LIN {X 0,Y 263.133,Z 902.515,A -85,B 0,C 180,E1 -18302.289,E2 -18302.289} C_VEL
LIN {X 0,Y 263.178,Z 902.512,A -85,B 0,C 180,E1 -18306.76,E2 -18306.76} C_VEL
LIN {X 0,Y 263.095,Z 902.525,A -85,B 0,C 180,E1 -18309.875,E2 -18309.875} C_VEL
LIN {X 0,Y 263.08,Z 902.529,A -85,B 0,C 180,E1 -18313.994,E2 -18313.994} C_VEL
LIN {X 0,Y 263.112,Z 902.522,A -85,B 0,C 180,E1 -18318.41,E2 -18318.41} C_VEL
LIN {X 0,Y 263.133,Z 902.519,A -85,B 0,C 180,E1 -18322.098,E2 -18322.098} C_VEL
LIN {X 0,Y 263.155,Z 902.516,A -85,B 0,C 180,E1 -18325.885,E2 -18325.885} C_VEL
LIN {X 0,Y 263.129,Z 902.516,A -85,B 0,C 180,E1 -18329.503,E2 -18329.503} C_VEL
LIN {X 0,Y 263.13,Z 902.521,A -85,B 0,C 180,E1 -18332.995,E2 -18332.995} C_VEL
LIN {X 0,Y 263.118,Z 902.52,A -85,B 0,C 180,E1 -18336.38,E2 -18336.38} C_VEL
LIN {X 0,Y 263.21,Z 902.507,A -85,B 0,C 180,E1 -18339.688,E2 -18339.688} C_VEL
LIN {X 0,Y 263.292,Z 902.498,A -85,B 0,C 180,E1 -18344.518,E2 -18344.518} C_VEL
LIN {X 0,Y 263.334,Z 902.493,A -85,B 0,C 180,E1 -18349.232,E2 -18349.232} C_VEL
LIN {X 0,Y 263.529,Z 902.469,A -85,B 0,C 180,E1 -18352.336,E2 -18352.336} C_VEL
LIN {X 0,Y 263.726,Z 902.443,A -85,B 0,C 180,E1 -18358.472,E2 -18358.472} C_VEL
LIN {X 0,Y 263.726,Z 902.445,A -85,B 0,C 180,E1 -18361.526,E2 -18361.526} C_VEL
LIN {X 0,Y 263.528,Z 902.467,A -85,B 0,C 180,E1 -18367.662,E2 -18367.662} C_VEL
LIN {X 0,Y 263.345,Z 902.494,A -85,B 0,C 180,E1 -18370.766,E2 -18370.766} C_VEL
LIN {X 0,Y 263.29,Z 902.496,A -85,B 0,C 180,E1 -18375.481,E2 -18375.481} C_VEL
LIN {X 0,Y 263.208,Z 902.509,A -85,B 0,C 180,E1 -18380.31,E2 -18380.31} C_VEL
LIN {X 0,Y 263.126,Z 902.52,A -85,B 0,C 180,E1 -18385.299,E2 -18385.299} C_VEL
LIN {X 0,Y 263.132,Z 902.518,A -85,B 0,C 180,E1 -18388.738,E2 -18388.738} C_VEL
LIN {X 0,Y 262.413,Z 902.609,A -85,B 0,C 180,E1 -18390.015,E2 -18390.015} C_VEL
LIN {X 0,Y 259.57,Z 902.961,A -85,B 0,C 180,E1 -18392.099,E2 -18392.099} C_VEL
LIN {X 0,Y 257.184,Z 903.26,A -85,B 0,C 180,E1 -18393.793,E2 -18393.793} C_VEL
LIN {X 0,Y 256.155,Z 903.386,A -85,B 0,C 180,E1 -18395.105,E2 -18395.105} C_VEL
LIN {X 0,Y 256.065,Z 903.395,A -85,B 0,C 180,E1 -18395.55,E2 -18395.55} C_VEL
LIN {X 0,Y 256.066,Z 903.399,A -85,B 0,C 180,E1 -18399.142,E2 -18399.142} C_VEL
LIN {X 0,Y 256.028,Z 903.402,A -85,B 0,C 180,E1 -18403.334,E2 -18403.334} C_VEL
LIN {X 0,Y 256.055,Z 903.402,A -85,B 0,C 180,E1 -18407.822,E2 -18407.822} C_VEL
LIN {X 0,Y 256.065,Z 903.398,A -85,B 0,C 180,E1 -18410.856,E2 -18410.856} C_VEL
LIN {X 0,Y 256.12,Z 903.39,A -85,B 0,C 180,E1 -18412.865,E2 -18412.865} C_VEL
LIN {X 0,Y 256.065,Z 903.401,A -85,B 0,C 180,E1 -18416.706,E2 -18416.706} C_VEL
LIN {X 0,Y 256.251,Z 903.416,A -85,B 0,C 180,E1 -18421.718,E2 -18421.718} C_VEL
LIN {X 0,Y 258.143,Z 913.925,A -85,B 0,C 180,E1 -18425.897,E2 -18425.897} C_VEL
LIN {X 0,Y 257.046,Z 922.563,A -85,B 0,C 180,E1 -18429.179,E2 -18429.179} C_VEL
LIN {X 0,Y 256.802,Z 924.586,A -85,B 0,C 180,E1 -18429.943,E2 -18429.943} C_VEL
LIN {X 0,Y 257.654,Z 940.89,A -85,B 0,C 180,E1 -18430.712,E2 -18430.712} C_VEL
LIN {X 0,Y 259.789,Z 963.766,A -85,B 0,C 180,E1 -18431.766,E2 -18431.766} C_VEL
LIN {X 0,Y 258.613,Z 1004.147,A -85,B 0,C 180,E1 -18433.572,E2 -18433.572} C_VEL
LIN {X 0,Y 257.814,Z 1016.929,A -85,B 0,C 180,E1 -18434.485,E2 -18434.485} C_VEL
LIN {X 0,Y 257.36,Z 1025.939,A -85,B 0,C 180,E1 -18435.368,E2 -18435.368} C_VEL
LIN {X 0,Y 256.718,Z 1035.432,A -85,B 0,C 180,E1 -18436.544,E2 -18436.544} C_VEL
LIN {X 0,Y 255.948,Z 1045.484,A -85,B 0,C 180,E1 -18438.115,E2 -18438.115} C_VEL
LIN {X 0,Y 255.437,Z 1053.431,A -85,B 0,C 180,E1 -18439.698,E2 -18439.698} C_VEL
LIN {X 0,Y 255.026,Z 1059.956,A -85,B 0,C 180,E1 -18441.282,E2 -18441.282} C_VEL
LIN {X 0,Y 254.757,Z 1065.381,A -85,B 0,C 180,E1 -18442.869,E2 -18442.869} C_VEL
LIN {X 0,Y 254.53,Z 1070.615,A -85,B 0,C 180,E1 -18444.755,E2 -18444.755} C_VEL
LIN {X 0,Y 254.336,Z 1075.116,A -85,B 0,C 180,E1 -18446.832,E2 -18446.832} C_VEL
LIN {X 0,Y 254.233,Z 1078.877,A -85,B 0,C 180,E1 -18449.208,E2 -18449.208} C_VEL
LIN {X 0,Y 254.094,Z 1081.168,A -85,B 0,C 180,E1 -18451.585,E2 -18451.585} C_VEL
LIN {X 0,Y 254.152,Z 1082.036,A -85,B 0,C 180,E1 -18453.17,E2 -18453.17} C_VEL
LIN {X 0,Y 254.131,Z 1082.299,A -85,B 0,C 180,E1 -18455.394,E2 -18455.394} C_VEL
LIN {X 0,Y 254.574,Z 1081.302,A -85,B 0,C 180,E1 -18457.934,E2 -18457.934} C_VEL
LIN {X 0,Y 255.122,Z 1080.076,A -85,B 0,C 180,E1 -18459.514,E2 -18459.514} C_VEL
LIN {X 0,Y 256.305,Z 1077.127,A -85,B 0,C 180,E1 -18461.867,E2 -18461.867} C_VEL
LIN {X 0,Y 257.32,Z 1074.54,A -85,B 0,C 180,E1 -18463.424,E2 -18463.424} C_VEL
LIN {X 0,Y 259.264,Z 1069.361,A -85,B 0,C 180,E1 -18465.728,E2 -18465.728} C_VEL
LIN {X 0,Y 261.247,Z 1063.88,A -85,B 0,C 180,E1 -18467.616,E2 -18467.616} C_VEL
LIN {X 0,Y 263.629,Z 1057.201,A -85,B 0,C 180,E1 -18469.465,E2 -18469.465} C_VEL
LIN {X 0,Y 266.42,Z 1048.971,A -85,B 0,C 180,E1 -18471.267,E2 -18471.267} C_VEL
LIN {X 0,Y 269.478,Z 1038.482,A -85,B 0,C 180,E1 -18473.029,E2 -18473.029} C_VEL
LIN {X 0,Y 272.034,Z 1029.452,A -85,B 0,C 180,E1 -18474.213,E2 -18474.213} C_VEL
LIN {X 0,Y 274.778,Z 1018.129,A -85,B 0,C 180,E1 -18475.367,E2 -18475.367} C_VEL
LIN {X 0,Y 276.831,Z 1007.471,A -85,B 0,C 180,E1 -18476.174,E2 -18476.174} C_VEL
LIN {X 0,Y 278.749,Z 994.655,A -85,B 0,C 180,E1 -18476.888,E2 -18476.888} C_VEL
LIN {X 0,Y 281.525,Z 969.653,A -85,B 0,C 180,E1 -18478.087,E2 -18478.087} C_VEL
LIN {X 0,Y 280.837,Z 960.401,A -85,B 0,C 180,E1 -18478.98,E2 -18478.98} C_VEL
LIN {X 0,Y 279.732,Z 952.159,A -85,B 0,C 180,E1 -18479.995,E2 -18479.995} C_VEL
LIN {X 0,Y 277.278,Z 946.159,A -85,B 0,C 180,E1 -18481.289,E2 -18481.289} C_VEL
LIN {X 0,Y 275.212,Z 941.618,A -85,B 0,C 180,E1 -18482.475,E2 -18482.475} C_VEL
LIN {X 0,Y 272.839,Z 936.693,A -85,B 0,C 180,E1 -18483.982,E2 -18483.982} C_VEL
LIN {X 0,Y 270.146,Z 931.863,A -85,B 0,C 180,E1 -18485.901,E2 -18485.901} C_VEL
LIN {X 0,Y 269.36,Z 930.385,A -85,B 0,C 180,E1 -18486.552,E2 -18486.552} C_VEL
LIN {X 0,Y 265.947,Z 924.786,A -85,B 0,C 180,E1 -18490.207,E2 -18490.207} C_VEL
LIN {X 0,Y 265.122,Z 922.952,A -85,B 0,C 180,E1 -18491.764,E2 -18491.764} C_VEL
LIN {X 0,Y 264.299,Z 921.573,A -85,B 0,C 180,E1 -18494.549,E2 -18494.549} C_VEL
LIN {X 0,Y 264.876,Z 921.163,A -85,B 0,C 180,E1 -18497.981,E2 -18497.981} C_VEL
LIN {X 0,Y 267.039,Z 924.13,A -85,B 0,C 180,E1 -18501.686,E2 -18501.686} C_VEL
LIN {X 0,Y 268.847,Z 925.751,A -85,B 0,C 180,E1 -18503.356,E2 -18503.356} C_VEL
LIN {X 0,Y 271.774,Z 929.696,A -85,B 0,C 180,E1 -18505.647,E2 -18505.647} C_VEL
LIN {X 0,Y 275.456,Z 935.246,A -85,B 0,C 180,E1 -18507.921,E2 -18507.921} C_VEL
LIN {X 0,Y 278.032,Z 939.659,A -85,B 0,C 180,E1 -18509.312,E2 -18509.312} C_VEL
LIN {X 0,Y 281.299,Z 945.577,A -85,B 0,C 180,E1 -18510.871,E2 -18510.871} C_VEL
LIN {X 0,Y 283.341,Z 950.251,A -85,B 0,C 180,E1 -18511.833,E2 -18511.833} C_VEL
LIN {X 0,Y 278.626,Z 988.353,A -85,B 0,C 180,E1 -18513.655,E2 -18513.655} C_VEL
LIN {X 0,Y 276.931,Z 999.245,A -85,B 0,C 180,E1 -18514.442,E2 -18514.442} C_VEL
LIN {X 0,Y 274.839,Z 1009.763,A -85,B 0,C 180,E1 -18515.448,E2 -18515.448} C_VEL
LIN {X 0,Y 272.517,Z 1019.531,A -85,B 0,C 180,E1 -18516.641,E2 -18516.641} C_VEL
LIN {X 0,Y 269.795,Z 1029.32,A -85,B 0,C 180,E1 -18518.211,E2 -18518.211} C_VEL
LIN {X 0,Y 267.014,Z 1038.1,A -85,B 0,C 180,E1 -18519.992,E2 -18519.992} C_VEL
LIN {X 0,Y 264.523,Z 1045.179,A -85,B 0,C 180,E1 -18521.81,E2 -18521.81} C_VEL
LIN {X 0,Y 262.291,Z 1050.771,A -85,B 0,C 180,E1 -18523.66,E2 -18523.66} C_VEL
LIN {X 0,Y 260.607,Z 1054.482,A -85,B 0,C 180,E1 -18525.156,E2 -18525.156} C_VEL
LIN {X 0,Y 258.571,Z 1058.706,A -85,B 0,C 180,E1 -18527.442,E2 -18527.442} C_VEL
LIN {X 0,Y 257.501,Z 1060.839,A -85,B 0,C 180,E1 -18528.987,E2 -18528.987} C_VEL
LIN {X 0,Y 256.624,Z 1062.359,A -85,B 0,C 180,E1 -18530.543,E2 -18530.543} C_VEL
LIN {X 0,Y 255.786,Z 1063.32,A -85,B 0,C 180,E1 -18532.104,E2 -18532.104} C_VEL
LIN {X 0,Y 255.092,Z 1063.796,A -85,B 0,C 180,E1 -18533.674,E2 -18533.674} C_VEL
LIN {X 0,Y 254.684,Z 1063.773,A -85,B 0,C 180,E1 -18535.252,E2 -18535.252} C_VEL
LIN {X 0,Y 254.42,Z 1063.24,A -85,B 0,C 180,E1 -18536.834,E2 -18536.834} C_VEL
LIN {X 0,Y 254.211,Z 1062.102,A -85,B 0,C 180,E1 -18538.417,E2 -18538.417} C_VEL
LIN {X 0,Y 254.09,Z 1059.449,A -85,B 0,C 180,E1 -18540.793,E2 -18540.793} C_VEL
LIN {X 0,Y 254.195,Z 1055.35,A -85,B 0,C 180,E1 -18543.171,E2 -18543.171} C_VEL
LIN {X 0,Y 254.272,Z 1050.813,A -85,B 0,C 180,E1 -18545.152,E2 -18545.152} C_VEL
LIN {X 0,Y 254.649,Z 1045.089,A -85,B 0,C 180,E1 -18547.135,E2 -18547.135} C_VEL
LIN {X 0,Y 255.093,Z 1037.972,A -85,B 0,C 180,E1 -18549.116,E2 -18549.116} C_VEL
LIN {X 0,Y 255.772,Z 1028.878,A -85,B 0,C 180,E1 -18551.09,E2 -18551.09} C_VEL
LIN {X 0,Y 256.352,Z 1021.061,A -85,B 0,C 180,E1 -18552.469,E2 -18552.469} C_VEL
LIN {X 0,Y 256.929,Z 1012.996,A -85,B 0,C 180,E1 -18553.647,E2 -18553.647} C_VEL
LIN {X 0,Y 257.62,Z 1003.027,A -85,B 0,C 180,E1 -18554.819,E2 -18554.819} C_VEL
LIN {X 0,Y 258.247,Z 990.644,A -85,B 0,C 180,E1 -18555.894,E2 -18555.894} C_VEL
LIN {X 0,Y 258.556,Z 981.199,A -85,B 0,C 180,E1 -18556.483,E2 -18556.483} C_VEL
LIN {X 0,Y 260.259,Z 930.177,A -85,B 0,C 180,E1 -18558.702,E2 -18558.702} C_VEL
LIN {X 0,Y 256.449,Z 904,A -85,B 0,C 180,E1 -18559.967,E2 -18559.967} C_VEL
LIN {X 0,Y 256.371,Z 903.35,A -85,B 0,C 180,E1 -18560.354,E2 -18560.354} C_VEL
LIN {X 0,Y 256.075,Z 903.397,A -85,B 0,C 180,E1 -18566.049,E2 -18566.049} C_VEL
LIN {X 0,Y 256.056,Z 903.399,A -85,B 0,C 180,E1 -18569.608,E2 -18569.608} C_VEL
LIN {X 0,Y 256.068,Z 903.401,A -85,B 0,C 180,E1 -18573.294,E2 -18573.294} C_VEL
LIN {X 0,Y 256.088,Z 903.397,A -85,B 0,C 180,E1 -18577.263,E2 -18577.263} C_VEL
LIN {X 0,Y 256.011,Z 903.404,A -85,B 0,C 180,E1 -18581.213,E2 -18581.213} C_VEL
LIN {X 0,Y 256.02,Z 903.405,A -85,B 0,C 180,E1 -18585.54,E2 -18585.54} C_VEL
LIN {X 0,Y 256.041,Z 903.4,A -85,B 0,C 180,E1 -18588.794,E2 -18588.794} C_VEL
LIN {X 0,Y 256.124,Z 903.392,A -85,B 0,C 180,E1 -18592.867,E2 -18592.867} C_VEL
LIN {X 0,Y 256.069,Z 903.398,A -85,B 0,C 180,E1 -18596.708,E2 -18596.708} C_VEL
LIN {X 0,Y 256.058,Z 903.401,A -85,B 0,C 180,E1 -18600.393,E2 -18600.393} C_VEL
LIN {X 0,Y 256.136,Z 903.393,A -85,B 0,C 180,E1 -18604.889,E2 -18604.889} C_VEL
LIN {X 0,Y 256.128,Z 903.394,A -85,B 0,C 180,E1 -18609.102,E2 -18609.102} C_VEL
LIN {X 0,Y 256.233,Z 903.376,A -85,B 0,C 180,E1 -18614.081,E2 -18614.081} C_VEL
LIN {X 0,Y 256.291,Z 903.37,A -85,B 0,C 180,E1 -18618.933,E2 -18618.933} C_VEL
LIN {X 0,Y 256.494,Z 903.346,A -85,B 0,C 180,E1 -18622.126,E2 -18622.126} C_VEL
LIN {X 0,Y 256.422,Z 903.352,A -85,B 0,C 180,E1 -18626.858,E2 -18626.858} C_VEL
LIN {X 0,Y 256.69,Z 903.321,A -85,B 0,C 180,E1 -18628.431,E2 -18628.431} C_VEL
LIN {X 0,Y 256.689,Z 903.321,A -85,B 0,C 180,E1 -18631.569,E2 -18631.569} C_VEL
LIN {X 0,Y 256.457,Z 903.352,A -85,B 0,C 180,E1 -18636.294,E2 -18636.294} C_VEL
LIN {X 0,Y 256.407,Z 903.355,A -85,B 0,C 180,E1 -18639.466,E2 -18639.466} C_VEL
LIN {X 0,Y 256.208,Z 903.38,A -85,B 0,C 180,E1 -18644.293,E2 -18644.293} C_VEL
LIN {X 0,Y 256.15,Z 903.388,A -85,B 0,C 180,E1 -18647.567,E2 -18647.567} C_VEL
LIN {X 0,Y 256.124,Z 903.393,A -85,B 0,C 180,E1 -18651.097,E2 -18651.097} C_VEL
LIN {X 0,Y 256.089,Z 903.398,A -85,B 0,C 180,E1 -18655.089,E2 -18655.089} C_VEL
LIN {X 0,Y 256.094,Z 903.395,A -85,B 0,C 180,E1 -18658.575,E2 -18658.575} C_VEL
LIN {X 0,Y 256.078,Z 903.396,A -85,B 0,C 180,E1 -18661.701,E2 -18661.701} C_VEL
LIN {X 0,Y 256.083,Z 903.397,A -85,B 0,C 180,E1 -18665.193,E2 -18665.193} C_VEL
LIN {X 0,Y 256.109,Z 903.395,A -85,B 0,C 180,E1 -18667.267,E2 -18667.267} C_VEL
LIN {X 0,Y 256.043,Z 903.399,A -85,B 0,C 180,E1 -18671.206,E2 -18671.206} C_VEL
LIN {X 0,Y 256.022,Z 903.405,A -85,B 0,C 180,E1 -18675.539,E2 -18675.539} C_VEL
LIN {X 0,Y 256.043,Z 903.4,A -85,B 0,C 180,E1 -18678.793,E2 -18678.793} C_VEL
LIN {X 0,Y 256.107,Z 903.393,A -85,B 0,C 180,E1 -18682.862,E2 -18682.862} C_VEL
LIN {X 0,Y 256.07,Z 903.4,A -85,B 0,C 180,E1 -18686.707,E2 -18686.707} C_VEL
LIN {X 0,Y 256.058,Z 903.399,A -85,B 0,C 180,E1 -18690.392,E2 -18690.392} C_VEL
LIN {X 0,Y 256.077,Z 903.396,A -85,B 0,C 180,E1 -18693.951,E2 -18693.951} C_VEL
LIN {X 0,Y 256.06,Z 903.399,A -85,B 0,C 180,E1 -18697.402,E2 -18697.402} C_VEL
LIN {X 0,Y 256.107,Z 903.393,A -85,B 0,C 180,E1 -18700.773,E2 -18700.773} C_VEL
LIN {X 0,Y 256.217,Z 903.379,A -85,B 0,C 180,E1 -18704.079,E2 -18704.079} C_VEL
LIN {X 0,Y 256.278,Z 903.37,A -85,B 0,C 180,E1 -18708.932,E2 -18708.932} C_VEL
LIN {X 0,Y 256.493,Z 903.346,A -85,B 0,C 180,E1 -18712.125,E2 -18712.125} C_VEL
LIN {X 0,Y 256.419,Z 903.352,A -85,B 0,C 180,E1 -18716.857,E2 -18716.857} C_VEL
LIN {X 0,Y 256.688,Z 903.32,A -85,B 0,C 180,E1 -18718.43,E2 -18718.43} C_VEL
LIN {X 0,Y 256.687,Z 903.322,A -85,B 0,C 180,E1 -18721.568,E2 -18721.568} C_VEL
LIN {X 0,Y 256.454,Z 903.352,A -85,B 0,C 180,E1 -18726.293,E2 -18726.293} C_VEL
LIN {X 0,Y 256.404,Z 903.355,A -85,B 0,C 180,E1 -18729.465,E2 -18729.465} C_VEL
LIN {X 0,Y 256.205,Z 903.382,A -85,B 0,C 180,E1 -18734.292,E2 -18734.292} C_VEL
LIN {X 0,Y 256.146,Z 903.387,A -85,B 0,C 180,E1 -18737.566,E2 -18737.566} C_VEL
LIN {X 0,Y 256.12,Z 903.395,A -85,B 0,C 180,E1 -18741.096,E2 -18741.096} C_VEL
LIN {X 0,Y 256.085,Z 903.398,A -85,B 0,C 180,E1 -18745.088,E2 -18745.088} C_VEL
LIN {X 0,Y 256.08,Z 903.396,A -85,B 0,C 180,E1 -18748.716,E2 -18748.716} C_VEL
LIN {X 0,Y 256.074,Z 903.399,A -85,B 0,C 180,E1 -18751.7,E2 -18751.7} C_VEL
LIN {X 0,Y 256.065,Z 903.395,A -85,B 0,C 180,E1 -18755.55,E2 -18755.55} C_VEL
LIN {X 0,Y 255.361,Z 903.486,A -85,B 0,C 180,E1 -18756.862,E2 -18756.862} C_VEL
LIN {X 0,Y 252.442,Z 903.85,A -85,B 0,C 180,E1 -18759,E2 -18759} C_VEL
LIN {X 0,Y 250.017,Z 904.151,A -85,B 0,C 180,E1 -18760.74,E2 -18760.74} C_VEL
LIN {X 0,Y 249.034,Z 904.275,A -85,B 0,C 180,E1 -18762.092,E2 -18762.092} C_VEL
LIN {X 0,Y 248.985,Z 904.278,A -85,B 0,C 180,E1 -18762.549,E2 -18762.549} C_VEL
LIN {X 0,Y 248.992,Z 904.279,A -85,B 0,C 180,E1 -18767.357,E2 -18767.357} C_VEL
LIN {X 0,Y 249.036,Z 904.276,A -85,B 0,C 180,E1 -18772.202,E2 -18772.202} C_VEL
LIN {X 0,Y 249.042,Z 904.272,A -85,B 0,C 180,E1 -18775.639,E2 -18775.639} C_VEL
LIN {X 0,Y 249.063,Z 904.27,A -85,B 0,C 180,E1 -18779.474,E2 -18779.474} C_VEL
LIN {X 0,Y 249.221,Z 904.386,A -85,B 0,C 180,E1 -18781.755,E2 -18781.755} C_VEL
LIN {X 0,Y 251.008,Z 913.787,A -85,B 0,C 180,E1 -18785.607,E2 -18785.607} C_VEL
LIN {X 0,Y 250.576,Z 918.515,A -85,B 0,C 180,E1 -18787.467,E2 -18787.467} C_VEL
LIN {X 0,Y 249.741,Z 924.538,A -85,B 0,C 180,E1 -18789.781,E2 -18789.781} C_VEL
LIN {X 0,Y 250.582,Z 941.022,A -85,B 0,C 180,E1 -18790.561,E2 -18790.561} C_VEL
LIN {X 0,Y 252.716,Z 964.072,A -85,B 0,C 180,E1 -18791.658,E2 -18791.658} C_VEL
LIN {X 0,Y 251.522,Z 1004.006,A -85,B 0,C 180,E1 -18793.513,E2 -18793.513} C_VEL
LIN {X 0,Y 250.741,Z 1016.613,A -85,B 0,C 180,E1 -18794.453,E2 -18794.453} C_VEL
LIN {X 0,Y 250.286,Z 1025.554,A -85,B 0,C 180,E1 -18795.361,E2 -18795.361} C_VEL
LIN {X 0,Y 249.63,Z 1034.982,A -85,B 0,C 180,E1 -18796.569,E2 -18796.569} C_VEL
LIN {X 0,Y 248.895,Z 1045.021,A -85,B 0,C 180,E1 -18798.187,E2 -18798.187} C_VEL
LIN {X 0,Y 248.369,Z 1052.947,A -85,B 0,C 180,E1 -18799.813,E2 -18799.813} C_VEL
LIN {X 0,Y 247.955,Z 1059.493,A -85,B 0,C 180,E1 -18801.442,E2 -18801.442} C_VEL
LIN {X 0,Y 247.675,Z 1065.579,A -85,B 0,C 180,E1 -18803.288,E2 -18803.288} C_VEL
LIN {X 0,Y 247.481,Z 1070.445,A -85,B 0,C 180,E1 -18805.112,E2 -18805.112} C_VEL
LIN {X 0,Y 247.336,Z 1073.949,A -85,B 0,C 180,E1 -18806.742,E2 -18806.742} C_VEL
LIN {X 0,Y 247.221,Z 1076.763,A -85,B 0,C 180,E1 -18808.371,E2 -18808.371} C_VEL
LIN {X 0,Y 247.214,Z 1078.945,A -85,B 0,C 180,E1 -18810,E2 -18810} C_VEL
LIN {X 0,Y 247.029,Z 1080.482,A -85,B 0,C 180,E1 -18811.63,E2 -18811.63} C_VEL
LIN {X 0,Y 247.084,Z 1081.422,A -85,B 0,C 180,E1 -18813.261,E2 -18813.261} C_VEL
LIN {X 0,Y 247.034,Z 1081.887,A -85,B 0,C 180,E1 -18815.302,E2 -18815.302} C_VEL
LIN {X 0,Y 247.526,Z 1081.253,A -85,B 0,C 180,E1 -18818.161,E2 -18818.161} C_VEL
LIN {X 0,Y 248.109,Z 1080.109,A -85,B 0,C 180,E1 -18819.785,E2 -18819.785} C_VEL
LIN {X 0,Y 249.372,Z 1077.508,A -85,B 0,C 180,E1 -18822.202,E2 -18822.202} C_VEL
LIN {X 0,Y 251.129,Z 1073.57,A -85,B 0,C 180,E1 -18824.588,E2 -18824.588} C_VEL
LIN {X 0,Y 252.5,Z 1070.287,A -85,B 0,C 180,E1 -18826.161,E2 -18826.161} C_VEL
LIN {X 0,Y 255.068,Z 1063.948,A -85,B 0,C 180,E1 -18828.473,E2 -18828.473} C_VEL
LIN {X 0,Y 257.629,Z 1057.311,A -85,B 0,C 180,E1 -18830.353,E2 -18830.353} C_VEL
LIN {X 0,Y 260.593,Z 1049.298,A -85,B 0,C 180,E1 -18832.183,E2 -18832.183} C_VEL
LIN {X 0,Y 263.889,Z 1039.169,A -85,B 0,C 180,E1 -18833.963,E2 -18833.963} C_VEL
LIN {X 0,Y 266.569,Z 1030.293,A -85,B 0,C 180,E1 -18835.159,E2 -18835.159} C_VEL
LIN {X 0,Y 269.459,Z 1019.526,A -85,B 0,C 180,E1 -18836.32,E2 -18836.32} C_VEL
LIN {X 0,Y 272.093,Z 1007.264,A -85,B 0,C 180,E1 -18837.288,E2 -18837.288} C_VEL
LIN {X 0,Y 274.032,Z 995.366,A -85,B 0,C 180,E1 -18837.977,E2 -18837.977} C_VEL
LIN {X 0,Y 276.931,Z 971.23,A -85,B 0,C 180,E1 -18839.157,E2 -18839.157} C_VEL
LIN {X 0,Y 276.42,Z 962.412,A -85,B 0,C 180,E1 -18840.076,E2 -18840.076} C_VEL
LIN {X 0,Y 275.567,Z 955.926,A -85,B 0,C 180,E1 -18840.917,E2 -18840.917} C_VEL
LIN {X 0,Y 273.306,Z 950.276,A -85,B 0,C 180,E1 -18842.274,E2 -18842.274} C_VEL
LIN {X 0,Y 271.796,Z 946.828,A -85,B 0,C 180,E1 -18843.219,E2 -18843.219} C_VEL
LIN {X 0,Y 269.843,Z 942.516,A -85,B 0,C 180,E1 -18844.587,E2 -18844.587} C_VEL
LIN {X 0,Y 266.957,Z 936.862,A -85,B 0,C 180,E1 -18846.928,E2 -18846.928} C_VEL
LIN {X 0,Y 263.725,Z 931.026,A -85,B 0,C 180,E1 -18850.821,E2 -18850.821} C_VEL
LIN {X 0,Y 263.187,Z 929.665,A -85,B 0,C 180,E1 -18852.067,E2 -18852.067} C_VEL
LIN {X 0,Y 262.475,Z 928.294,A -85,B 0,C 180,E1 -18855.015,E2 -18855.015} C_VEL
LIN {X 0,Y 263.117,Z 928.175,A -85,B 0,C 180,E1 -18858.106,E2 -18858.106} C_VEL
LIN {X 0,Y 265.134,Z 930.965,A -85,B 0,C 180,E1 -18861.604,E2 -18861.604} C_VEL
LIN {X 0,Y 266.7,Z 932.504,A -85,B 0,C 180,E1 -18863.112,E2 -18863.112} C_VEL
LIN {X 0,Y 269.742,Z 936.883,A -85,B 0,C 180,E1 -18865.617,E2 -18865.617} C_VEL
LIN {X 0,Y 272.633,Z 941.5,A -85,B 0,C 180,E1 -18867.502,E2 -18867.502} C_VEL
LIN {X 0,Y 275.37,Z 946.378,A -85,B 0,C 180,E1 -18869.053,E2 -18869.053} C_VEL
LIN {X 0,Y 278.517,Z 952.741,A -85,B 0,C 180,E1 -18870.672,E2 -18870.672} C_VEL
LIN {X 0,Y 278.768,Z 953.348,A -85,B 0,C 180,E1 -18870.801,E2 -18870.801} C_VEL
LIN {X 0,Y 273.886,Z 989.769,A -85,B 0,C 180,E1 -18872.595,E2 -18872.595} C_VEL
LIN {X 0,Y 272.158,Z 999.794,A -85,B 0,C 180,E1 -18873.342,E2 -18873.342} C_VEL
LIN {X 0,Y 269.921,Z 1010.106,A -85,B 0,C 180,E1 -18874.351,E2 -18874.351} C_VEL
LIN {X 0,Y 267.409,Z 1019.743,A -85,B 0,C 180,E1 -18875.548,E2 -18875.548} C_VEL
LIN {X 0,Y 264.801,Z 1028.684,A -85,B 0,C 180,E1 -18876.954,E2 -18876.954} C_VEL
LIN {X 0,Y 262.369,Z 1035.94,A -85,B 0,C 180,E1 -18878.389,E2 -18878.389} C_VEL
LIN {X 0,Y 260.077,Z 1042.023,A -85,B 0,C 180,E1 -18879.847,E2 -18879.847} C_VEL
LIN {X 0,Y 257.515,Z 1048.284,A -85,B 0,C 180,E1 -18881.709,E2 -18881.709} C_VEL
LIN {X 0,Y 255.67,Z 1052.427,A -85,B 0,C 180,E1 -18883.225,E2 -18883.225} C_VEL
LIN {X 0,Y 253.904,Z 1055.889,A -85,B 0,C 180,E1 -18884.755,E2 -18884.755} C_VEL
LIN {X 0,Y 251.731,Z 1059.801,A -85,B 0,C 180,E1 -18887.095,E2 -18887.095} C_VEL
LIN {X 0,Y 250.121,Z 1062.545,A -85,B 0,C 180,E1 -18889.559,E2 -18889.559} C_VEL
LIN {X 0,Y 248.809,Z 1063.966,A -85,B 0,C 180,E1 -18891.882,E2 -18891.882} C_VEL
LIN {X 0,Y 248.062,Z 1064.228,A -85,B 0,C 180,E1 -18893.494,E2 -18893.494} C_VEL
LIN {X 0,Y 247.621,Z 1063.995,A -85,B 0,C 180,E1 -18895.116,E2 -18895.116} C_VEL
LIN {X 0,Y 247.337,Z 1063.284,A -85,B 0,C 180,E1 -18896.743,E2 -18896.743} C_VEL
LIN {X 0,Y 247.141,Z 1062.058,A -85,B 0,C 180,E1 -18898.371,E2 -18898.371} C_VEL
LIN {X 0,Y 247.019,Z 1059.063,A -85,B 0,C 180,E1 -18900.816,E2 -18900.816} C_VEL
LIN {X 0,Y 247.106,Z 1056.406,A -85,B 0,C 180,E1 -18902.446,E2 -18902.446} C_VEL
LIN {X 0,Y 247.172,Z 1052.073,A -85,B 0,C 180,E1 -18904.485,E2 -18904.485} C_VEL
LIN {X 0,Y 247.432,Z 1046.559,A -85,B 0,C 180,E1 -18906.525,E2 -18906.525} C_VEL
LIN {X 0,Y 247.906,Z 1039.671,A -85,B 0,C 180,E1 -18908.56,E2 -18908.56} C_VEL
LIN {X 0,Y 248.496,Z 1031.079,A -85,B 0,C 180,E1 -18910.594,E2 -18910.594} C_VEL
LIN {X 0,Y 249.126,Z 1022.37,A -85,B 0,C 180,E1 -18912.216,E2 -18912.216} C_VEL
LIN {X 0,Y 249.726,Z 1014.502,A -85,B 0,C 180,E1 -18913.426,E2 -18913.426} C_VEL
LIN {X 0,Y 250.355,Z 1004.831,A -85,B 0,C 180,E1 -18914.635,E2 -18914.635} C_VEL
LIN {X 0,Y 251.056,Z 993.496,A -85,B 0,C 180,E1 -18915.736,E2 -18915.736} C_VEL
LIN {X 0,Y 251.439,Z 981.374,A -85,B 0,C 180,E1 -18916.545,E2 -18916.545} C_VEL
LIN {X 0,Y 252.953,Z 937.801,A -85,B 0,C 180,E1 -18918.538,E2 -18918.538} C_VEL
LIN {X 0,Y 253.031,Z 929.686,A -85,B 0,C 180,E1 -18918.9,E2 -18918.9} C_VEL
LIN {X 0,Y 249.336,Z 904.287,A -85,B 0,C 180,E1 -18920.167,E2 -18920.167} C_VEL
LIN {X 0,Y 249.048,Z 904.275,A -85,B 0,C 180,E1 -18925.442,E2 -18925.442} C_VEL
LIN {X 0,Y 249.037,Z 904.275,A -85,B 0,C 180,E1 -18928.974,E2 -18928.974} C_VEL
LIN {X 0,Y 249.029,Z 904.274,A -85,B 0,C 180,E1 -18932.427,E2 -18932.427} C_VEL
LIN {X 0,Y 249.012,Z 904.276,A -85,B 0,C 180,E1 -18936.35,E2 -18936.35} C_VEL
LIN {X 0,Y 248.973,Z 904.281,A -85,B 0,C 180,E1 -18940.486,E2 -18940.486} C_VEL
LIN {X 0,Y 248.964,Z 904.282,A -85,B 0,C 180,E1 -18944.889,E2 -18944.889} C_VEL
LIN {X 0,Y 248.995,Z 904.277,A -85,B 0,C 180,E1 -18947.359,E2 -18947.359} C_VEL
LIN {X 0,Y 249.039,Z 904.277,A -85,B 0,C 180,E1 -18952.203,E2 -18952.203} C_VEL
LIN {X 0,Y 249.046,Z 904.272,A -85,B 0,C 180,E1 -18955.64,E2 -18955.64} C_VEL
LIN {X 0,Y 249.005,Z 904.277,A -85,B 0,C 180,E1 -18959.467,E2 -18959.467} C_VEL
LIN {X 0,Y 249.038,Z 904.275,A -85,B 0,C 180,E1 -18963.158,E2 -18963.158} C_VEL
LIN {X 0,Y 249.055,Z 904.272,A -85,B 0,C 180,E1 -18966.73,E2 -18966.73} C_VEL
LIN {X 0,Y 249.06,Z 904.27,A -85,B 0,C 180,E1 -18970.208,E2 -18970.208} C_VEL
LIN {X 0,Y 249.162,Z 904.259,A -85,B 0,C 180,E1 -18973.617,E2 -18973.617} C_VEL
LIN {X 0,Y 249.19,Z 904.253,A -85,B 0,C 180,E1 -18976.96,E2 -18976.96} C_VEL
LIN {X 0,Y 249.39,Z 904.23,A -85,B 0,C 180,E1 -18980.52,E2 -18980.52} C_VEL
LIN {X 0,Y 249.431,Z 904.227,A -85,B 0,C 180,E1 -18983.529,E2 -18983.529} C_VEL
LIN {X 0,Y 249.65,Z 904.199,A -85,B 0,C 180,E1 -18988.387,E2 -18988.387} C_VEL
LIN {X 0,Y 249.65,Z 904.199,A -85,B 0,C 180,E1 -18991.613,E2 -18991.613} C_VEL
LIN {X 0,Y 249.431,Z 904.227,A -85,B 0,C 180,E1 -18996.472,E2 -18996.472} C_VEL
LIN {X 0,Y 249.338,Z 904.237,A -85,B 0,C 180,E1 -18999.737,E2 -18999.737} C_VEL
LIN {X 0,Y 249.152,Z 904.261,A -85,B 0,C 180,E1 -19004.707,E2 -19004.707} C_VEL
LIN {X 0,Y 249.082,Z 904.268,A -85,B 0,C 180,E1 -19008.082,E2 -19008.082} C_VEL
LIN {X 0,Y 249.047,Z 904.271,A -85,B 0,C 180,E1 -19011.522,E2 -19011.522} C_VEL
LIN {X 0,Y 249.051,Z 904.274,A -85,B 0,C 180,E1 -19015.441,E2 -19015.441} C_VEL
LIN {X 0,Y 249.04,Z 904.276,A -85,B 0,C 180,E1 -19018.973,E2 -19018.973} C_VEL
LIN {X 0,Y 249.032,Z 904.271,A -85,B 0,C 180,E1 -19022.426,E2 -19022.426} C_VEL
LIN {X 0,Y 249.028,Z 904.275,A -85,B 0,C 180,E1 -19026.346,E2 -19026.346} C_VEL
LIN {X 0,Y 248.988,Z 904.278,A -85,B 0,C 180,E1 -19030.482,E2 -19030.482} C_VEL
LIN {X 0,Y 248.987,Z 904.278,A -85,B 0,C 180,E1 -19032.786,E2 -19032.786} C_VEL
LIN {X 0,Y 248.997,Z 904.279,A -85,B 0,C 180,E1 -19037.357,E2 -19037.357} C_VEL
LIN {X 0,Y 249.047,Z 904.274,A -85,B 0,C 180,E1 -19042.2,E2 -19042.2} C_VEL
LIN {X 0,Y 249.047,Z 904.272,A -85,B 0,C 180,E1 -19045.639,E2 -19045.639} C_VEL
LIN {X 0,Y 249.006,Z 904.275,A -85,B 0,C 180,E1 -19049.466,E2 -19049.466} C_VEL
LIN {X 0,Y 249.025,Z 904.277,A -85,B 0,C 180,E1 -19053.156,E2 -19053.156} C_VEL
LIN {X 0,Y 249.009,Z 904.28,A -85,B 0,C 180,E1 -19056.725,E2 -19056.725} C_VEL
LIN {X 0,Y 249.044,Z 904.271,A -85,B 0,C 180,E1 -19060.205,E2 -19060.205} C_VEL
LIN {X 0,Y 249.161,Z 904.26,A -85,B 0,C 180,E1 -19063.616,E2 -19063.616} C_VEL
LIN {X 0,Y 249.223,Z 904.247,A -85,B 0,C 180,E1 -19068.614,E2 -19068.614} C_VEL
LIN {X 0,Y 249.434,Z 904.227,A -85,B 0,C 180,E1 -19071.9,E2 -19071.9} C_VEL
LIN {X 0,Y 249.251,Z 904.247,A -85,B 0,C 180,E1 -19075.147,E2 -19075.147} C_VEL
LIN {X 0,Y 249.648,Z 904.197,A -85,B 0,C 180,E1 -19078.386,E2 -19078.386} C_VEL
LIN {X 0,Y 249.648,Z 904.199,A -85,B 0,C 180,E1 -19081.612,E2 -19081.612} C_VEL
LIN {X 0,Y 249.426,Z 904.226,A -85,B 0,C 180,E1 -19086.471,E2 -19086.471} C_VEL
LIN {X 0,Y 249.335,Z 904.236,A -85,B 0,C 180,E1 -19089.736,E2 -19089.736} C_VEL
LIN {X 0,Y 249.149,Z 904.262,A -85,B 0,C 180,E1 -19094.706,E2 -19094.706} C_VEL
LIN {X 0,Y 249.078,Z 904.267,A -85,B 0,C 180,E1 -19098.081,E2 -19098.081} C_VEL
LIN {X 0,Y 249.044,Z 904.273,A -85,B 0,C 180,E1 -19101.521,E2 -19101.521} C_VEL
LIN {X 0,Y 249.048,Z 904.272,A -85,B 0,C 180,E1 -19105.44,E2 -19105.44} C_VEL
LIN {X 0,Y 249.036,Z 904.276,A -85,B 0,C 180,E1 -19108.973,E2 -19108.973} C_VEL
LIN {X 0,Y 249.028,Z 904.274,A -85,B 0,C 180,E1 -19112.425,E2 -19112.425} C_VEL
LIN {X 0,Y 249.024,Z 904.275,A -85,B 0,C 180,E1 -19116.346,E2 -19116.346} C_VEL
LIN {X 0,Y 248.984,Z 904.28,A -85,B 0,C 180,E1 -19120.482,E2 -19120.482} C_VEL
LIN {X 0,Y 248.985,Z 904.278,A -85,B 0,C 180,E1 -19122.549,E2 -19122.549} C_VEL
LIN {X 0,Y 248.723,Z 904.316,A -85,B 0,C 180,E1 -19123.451,E2 -19123.451} C_VEL
LIN {X 0,Y 247.401,Z 904.484,A -85,B 0,C 180,E1 -19124.784,E2 -19124.784} C_VEL
LIN {X 0,Y 243.028,Z 905.025,A -85,B 0,C 180,E1 -19127.889,E2 -19127.889} C_VEL
LIN {X 0,Y 241.986,Z 905.152,A -85,B 0,C 180,E1 -19129.28,E2 -19129.28} C_VEL
LIN {X 0,Y 241.914,Z 905.161,A -85,B 0,C 180,E1 -19129.752,E2 -19129.752} C_VEL
LIN {X 0,Y 241.979,Z 905.154,A -85,B 0,C 180,E1 -19132.416,E2 -19132.416} C_VEL
LIN {X 0,Y 241.978,Z 905.157,A -85,B 0,C 180,E1 -19136.507,E2 -19136.507} C_VEL
LIN {X 0,Y 242.173,Z 905.17,A -85,B 0,C 180,E1 -19141.744,E2 -19141.744} C_VEL
LIN {X 0,Y 243.945,Z 914.704,A -85,B 0,C 180,E1 -19145.761,E2 -19145.761} C_VEL
LIN {X 0,Y 242.708,Z 924.098,A -85,B 0,C 180,E1 -19149.556,E2 -19149.556} C_VEL
LIN {X 0,Y 243.507,Z 941.425,A -85,B 0,C 180,E1 -19150.431,E2 -19150.431} C_VEL
LIN {X 0,Y 245.614,Z 964.199,A -85,B 0,C 180,E1 -19151.557,E2 -19151.557} C_VEL
LIN {X 0,Y 244.441,Z 1003.975,A -85,B 0,C 180,E1 -19153.505,E2 -19153.505} C_VEL
LIN {X 0,Y 243.698,Z 1015.899,A -85,B 0,C 180,E1 -19154.421,E2 -19154.421} C_VEL
LIN {X 0,Y 243.108,Z 1026.626,A -85,B 0,C 180,E1 -19155.561,E2 -19155.561} C_VEL
LIN {X 0,Y 242.368,Z 1037.225,A -85,B 0,C 180,E1 -19157.013,E2 -19157.013} C_VEL
LIN {X 0,Y 241.73,Z 1046.577,A -85,B 0,C 180,E1 -19158.682,E2 -19158.682} C_VEL
LIN {X 0,Y 241.189,Z 1054.188,A -85,B 0,C 180,E1 -19160.354,E2 -19160.354} C_VEL
LIN {X 0,Y 240.841,Z 1060.646,A -85,B 0,C 180,E1 -19162.074,E2 -19162.074} C_VEL
LIN {X 0,Y 240.572,Z 1066.61,A -85,B 0,C 180,E1 -19164.028,E2 -19164.028} C_VEL
LIN {X 0,Y 240.332,Z 1072.714,A -85,B 0,C 180,E1 -19166.647,E2 -19166.647} C_VEL
LIN {X 0,Y 240.204,Z 1075.71,A -85,B 0,C 180,E1 -19168.323,E2 -19168.323} C_VEL
LIN {X 0,Y 240.187,Z 1078.017,A -85,B 0,C 180,E1 -19170,E2 -19170} C_VEL
LIN {X 0,Y 239.979,Z 1079.659,A -85,B 0,C 180,E1 -19171.678,E2 -19171.678} C_VEL
LIN {X 0,Y 240.016,Z 1080.796,A -85,B 0,C 180,E1 -19173.357,E2 -19173.357} C_VEL
LIN {X 0,Y 239.949,Z 1081.433,A -85,B 0,C 180,E1 -19175.23,E2 -19175.23} C_VEL
LIN {X 0,Y 240.132,Z 1081.546,A -85,B 0,C 180,E1 -19176.723,E2 -19176.723} C_VEL
LIN {X 0,Y 240.486,Z 1081.07,A -85,B 0,C 180,E1 -19178.402,E2 -19178.402} C_VEL
LIN {X 0,Y 241.116,Z 1080.108,A -85,B 0,C 180,E1 -19180.072,E2 -19180.072} C_VEL
LIN {X 0,Y 241.927,Z 1078.669,A -85,B 0,C 180,E1 -19181.733,E2 -19181.733} C_VEL
LIN {X 0,Y 243.606,Z 1075.504,A -85,B 0,C 180,E1 -19184.195,E2 -19184.195} C_VEL
LIN {X 0,Y 245.756,Z 1071.075,A -85,B 0,C 180,E1 -19186.617,E2 -19186.617} C_VEL
LIN {X 0,Y 248.466,Z 1065.252,A -85,B 0,C 180,E1 -19188.983,E2 -19188.983} C_VEL
LIN {X 0,Y 251.141,Z 1059.076,A -85,B 0,C 180,E1 -19190.904,E2 -19190.904} C_VEL
LIN {X 0,Y 254.234,Z 1051.429,A -85,B 0,C 180,E1 -19192.769,E2 -19192.769} C_VEL
LIN {X 0,Y 256.952,Z 1044.094,A -85,B 0,C 180,E1 -19194.222,E2 -19194.222} C_VEL
LIN {X 0,Y 259.576,Z 1036.523,A -85,B 0,C 180,E1 -19195.456,E2 -19195.456} C_VEL
LIN {X 0,Y 262.916,Z 1025.948,A -85,B 0,C 180,E1 -19196.813,E2 -19196.813} C_VEL
LIN {X 0,Y 266.073,Z 1013.731,A -85,B 0,C 180,E1 -19197.959,E2 -19197.959} C_VEL
LIN {X 0,Y 268.686,Z 1001.405,A -85,B 0,C 180,E1 -19198.83,E2 -19198.83} C_VEL
LIN {X 0,Y 272.604,Z 972.743,A -85,B 0,C 180,E1 -19200.299,E2 -19200.299} C_VEL
LIN {X 0,Y 272.102,Z 963.055,A -85,B 0,C 180,E1 -19201.393,E2 -19201.393} C_VEL
LIN {X 0,Y 271.71,Z 960.257,A -85,B 0,C 180,E1 -19201.813,E2 -19201.813} C_VEL
LIN {X 0,Y 269.175,Z 953.389,A -85,B 0,C 180,E1 -19203.546,E2 -19203.546} C_VEL
LIN {X 0,Y 266.865,Z 948.177,A -85,B 0,C 180,E1 -19205.275,E2 -19205.275} C_VEL
LIN {X 0,Y 264.462,Z 943.1,A -85,B 0,C 180,E1 -19207.466,E2 -19207.466} C_VEL
LIN {X 0,Y 261.65,Z 937.567,A -85,B 0,C 180,E1 -19211.229,E2 -19211.229} C_VEL
LIN {X 0,Y 261.299,Z 936.438,A -85,B 0,C 180,E1 -19212.253,E2 -19212.253} C_VEL
LIN {X 0,Y 260.67,Z 935.072,A -85,B 0,C 180,E1 -19215.494,E2 -19215.494} C_VEL
LIN {X 0,Y 261.303,Z 935.107,A -85,B 0,C 180,E1 -19218.113,E2 -19218.113} C_VEL
LIN {X 0,Y 263.434,Z 937.992,A -85,B 0,C 180,E1 -19221.76,E2 -19221.76} C_VEL
LIN {X 0,Y 264.49,Z 939.125,A -85,B 0,C 180,E1 -19222.8,E2 -19222.8} C_VEL
LIN {X 0,Y 267.108,Z 943.061,A -85,B 0,C 180,E1 -19225.107,E2 -19225.107} C_VEL
LIN {X 0,Y 269.817,Z 947.654,A -85,B 0,C 180,E1 -19227.031,E2 -19227.031} C_VEL
LIN {X 0,Y 271.839,Z 951.496,A -85,B 0,C 180,E1 -19228.303,E2 -19228.303} C_VEL
LIN {X 0,Y 274.331,Z 956.755,A -85,B 0,C 180,E1 -19229.744,E2 -19229.744} C_VEL
LIN {X 0,Y 269.81,Z 988.428,A -85,B 0,C 180,E1 -19231.322,E2 -19231.322} C_VEL
LIN {X 0,Y 267.935,Z 998.73,A -85,B 0,C 180,E1 -19232.04,E2 -19232.04} C_VEL
LIN {X 0,Y 265.161,Z 1010.702,A -85,B 0,C 180,E1 -19233.22,E2 -19233.22} C_VEL
LIN {X 0,Y 262.493,Z 1020.35,A -85,B 0,C 180,E1 -19234.423,E2 -19234.423} C_VEL
LIN {X 0,Y 259.331,Z 1030.073,A -85,B 0,C 180,E1 -19236.015,E2 -19236.015} C_VEL
LIN {X 0,Y 256.115,Z 1038.677,A -85,B 0,C 180,E1 -19237.833,E2 -19237.833} C_VEL
LIN {X 0,Y 253.151,Z 1045.762,A -85,B 0,C 180,E1 -19239.695,E2 -19239.695} C_VEL
LIN {X 0,Y 250.025,Z 1052.291,A -85,B 0,C 180,E1 -19241.99,E2 -19241.99} C_VEL
LIN {X 0,Y 247.194,Z 1057.306,A -85,B 0,C 180,E1 -19244.331,E2 -19244.331} C_VEL
LIN {X 0,Y 244.922,Z 1060.973,A -85,B 0,C 180,E1 -19246.73,E2 -19246.73} C_VEL
LIN {X 0,Y 243.213,Z 1063.386,A -85,B 0,C 180,E1 -19249.259,E2 -19249.259} C_VEL
LIN {X 0,Y 241.813,Z 1064.483,A -85,B 0,C 180,E1 -19251.645,E2 -19251.645} C_VEL
LIN {X 0,Y 241.037,Z 1064.65,A -85,B 0,C 180,E1 -19253.303,E2 -19253.303} C_VEL
LIN {X 0,Y 240.563,Z 1064.209,A -85,B 0,C 180,E1 -19254.973,E2 -19254.973} C_VEL
LIN {X 0,Y 240.257,Z 1063.283,A -85,B 0,C 180,E1 -19256.647,E2 -19256.647} C_VEL
LIN {X 0,Y 240.073,Z 1061.87,A -85,B 0,C 180,E1 -19258.323,E2 -19258.323} C_VEL
LIN {X 0,Y 239.95,Z 1058.649,A -85,B 0,C 180,E1 -19260.84,E2 -19260.84} C_VEL
LIN {X 0,Y 240.04,Z 1055.767,A -85,B 0,C 180,E1 -19262.518,E2 -19262.518} C_VEL
LIN {X 0,Y 240.116,Z 1050.142,A -85,B 0,C 180,E1 -19265.038,E2 -19265.038} C_VEL
LIN {X 0,Y 240.587,Z 1042.759,A -85,B 0,C 180,E1 -19267.554,E2 -19267.554} C_VEL
LIN {X 0,Y 240.987,Z 1036.569,A -85,B 0,C 180,E1 -19269.231,E2 -19269.231} C_VEL
LIN {X 0,Y 241.626,Z 1028.081,A -85,B 0,C 180,E1 -19271.111,E2 -19271.111} C_VEL
LIN {X 0,Y 242.312,Z 1018.754,A -85,B 0,C 180,E1 -19272.778,E2 -19272.778} C_VEL
LIN {X 0,Y 243.056,Z 1008.359,A -85,B 0,C 180,E1 -19274.229,E2 -19274.229} C_VEL
LIN {X 0,Y 243.607,Z 998.885,A -85,B 0,C 180,E1 -19275.264,E2 -19275.264} C_VEL
LIN {X 0,Y 244.058,Z 989.149,A -85,B 0,C 180,E1 -19276.092,E2 -19276.092} C_VEL
LIN {X 0,Y 244.545,Z 977.464,A -85,B 0,C 180,E1 -19276.81,E2 -19276.81} C_VEL
LIN {X 0,Y 246.008,Z 930.716,A -85,B 0,C 180,E1 -19279.002,E2 -19279.002} C_VEL
LIN {X 0,Y 242.443,Z 905.992,A -85,B 0,C 180,E1 -19280.253,E2 -19280.253} C_VEL
LIN {X 0,Y 242.273,Z 905.106,A -85,B 0,C 180,E1 -19280.372,E2 -19280.372} C_VEL
LIN {X 0,Y 241.988,Z 905.152,A -85,B 0,C 180,E1 -19285.827,E2 -19285.827} C_VEL
LIN {X 0,Y 241.97,Z 905.154,A -85,B 0,C 180,E1 -19289.589,E2 -19289.589} C_VEL
LIN {X 0,Y 241.981,Z 905.157,A -85,B 0,C 180,E1 -19293.494,E2 -19293.494} C_VEL
LIN {X 0,Y 241.966,Z 905.157,A -85,B 0,C 180,E1 -19297.587,E2 -19297.587} C_VEL
LIN {X 0,Y 241.907,Z 905.166,A -85,B 0,C 180,E1 -19301.93,E2 -19301.93} C_VEL
LIN {X 0,Y 241.911,Z 905.161,A -85,B 0,C 180,E1 -19306.579,E2 -19306.579} C_VEL
LIN {X 0,Y 241.993,Z 905.151,A -85,B 0,C 180,E1 -19311.643,E2 -19311.643} C_VEL
LIN {X 0,Y 241.981,Z 905.156,A -85,B 0,C 180,E1 -19314.488,E2 -19314.488} C_VEL
LIN {X 0,Y 241.956,Z 905.156,A -85,B 0,C 180,E1 -19318.477,E2 -19318.477} C_VEL
LIN {X 0,Y 241.971,Z 905.155,A -85,B 0,C 180,E1 -19322.308,E2 -19322.308} C_VEL
LIN {X 0,Y 242.027,Z 905.145,A -85,B 0,C 180,E1 -19326.013,E2 -19326.013} C_VEL
LIN {X 0,Y 241.995,Z 905.152,A -85,B 0,C 180,E1 -19329.605,E2 -19329.605} C_VEL
LIN {X 0,Y 242.118,Z 905.139,A -85,B 0,C 180,E1 -19333.319,E2 -19333.319} C_VEL
LIN {X 0,Y 242.168,Z 905.129,A -85,B 0,C 180,E1 -19338.279,E2 -19338.279} C_VEL
LIN {X 0,Y 242.389,Z 905.106,A -85,B 0,C 180,E1 -19341.665,E2 -19341.665} C_VEL
LIN {X 0,Y 242.404,Z 905.101,A -85,B 0,C 180,E1 -19343.341,E2 -19343.341} C_VEL
LIN {X 0,Y 242.609,Z 905.076,A -85,B 0,C 180,E1 -19348.34,E2 -19348.34} C_VEL
LIN {X 0,Y 242.609,Z 905.076,A -85,B 0,C 180,E1 -19351.66,E2 -19351.66} C_VEL
LIN {X 0,Y 242.403,Z 905.101,A -85,B 0,C 180,E1 -19356.66,E2 -19356.66} C_VEL
LIN {X 0,Y 242.266,Z 905.119,A -85,B 0,C 180,E1 -19360.024,E2 -19360.024} C_VEL
LIN {X 0,Y 242.11,Z 905.137,A -85,B 0,C 180,E1 -19365.145,E2 -19365.145} C_VEL
LIN {X 0,Y 242.02,Z 905.151,A -85,B 0,C 180,E1 -19368.629,E2 -19368.629} C_VEL
LIN {X 0,Y 241.977,Z 905.151,A -85,B 0,C 180,E1 -19372.184,E2 -19372.184} C_VEL
LIN {X 0,Y 241.991,Z 905.151,A -85,B 0,C 180,E1 -19375.826,E2 -19375.826} C_VEL
LIN {X 0,Y 241.973,Z 905.155,A -85,B 0,C 180,E1 -19379.588,E2 -19379.588} C_VEL
LIN {X 0,Y 241.984,Z 905.154,A -85,B 0,C 180,E1 -19383.493,E2 -19383.493} C_VEL
LIN {X 0,Y 241.984,Z 905.156,A -85,B 0,C 180,E1 -19387.583,E2 -19387.583} C_VEL
LIN {X 0,Y 241.922,Z 905.161,A -85,B 0,C 180,E1 -19391.926,E2 -19391.926} C_VEL
LIN {X 0,Y 241.913,Z 905.162,A -85,B 0,C 180,E1 -19396.577,E2 -19396.577} C_VEL
LIN {X 0,Y 241.997,Z 905.148,A -85,B 0,C 180,E1 -19401.641,E2 -19401.641} C_VEL
LIN {X 0,Y 241.979,Z 905.157,A -85,B 0,C 180,E1 -19404.487,E2 -19404.487} C_VEL
LIN {X 0,Y 241.957,Z 905.159,A -85,B 0,C 180,E1 -19408.476,E2 -19408.476} C_VEL
LIN {X 0,Y 241.964,Z 905.155,A -85,B 0,C 180,E1 -19412.306,E2 -19412.306} C_VEL
LIN {X 0,Y 241.961,Z 905.155,A -85,B 0,C 180,E1 -19416.005,E2 -19416.005} C_VEL
LIN {X 0,Y 241.985,Z 905.151,A -85,B 0,C 180,E1 -19419.602,E2 -19419.602} C_VEL
LIN {X 0,Y 242.109,Z 905.141,A -85,B 0,C 180,E1 -19423.324,E2 -19423.324} C_VEL
LIN {X 0,Y 242.157,Z 905.127,A -85,B 0,C 180,E1 -19428.277,E2 -19428.277} C_VEL
LIN {X 0,Y 242.384,Z 905.107,A -85,B 0,C 180,E1 -19431.663,E2 -19431.663} C_VEL
LIN {X 0,Y 242.401,Z 905.102,A -85,B 0,C 180,E1 -19433.339,E2 -19433.339} C_VEL
LIN {X 0,Y 242.607,Z 905.074,A -85,B 0,C 180,E1 -19438.339,E2 -19438.339} C_VEL
LIN {X 0,Y 242.607,Z 905.076,A -85,B 0,C 180,E1 -19441.659,E2 -19441.659} C_VEL
LIN {X 0,Y 242.396,Z 905.1,A -85,B 0,C 180,E1 -19446.659,E2 -19446.659} C_VEL
LIN {X 0,Y 242.263,Z 905.118,A -85,B 0,C 180,E1 -19450.023,E2 -19450.023} C_VEL
LIN {X 0,Y 242.107,Z 905.135,A -85,B 0,C 180,E1 -19455.144,E2 -19455.144} C_VEL
LIN {X 0,Y 242.017,Z 905.15,A -85,B 0,C 180,E1 -19458.628,E2 -19458.628} C_VEL
LIN {X 0,Y 241.974,Z 905.153,A -85,B 0,C 180,E1 -19462.183,E2 -19462.183} C_VEL
LIN {X 0,Y 241.987,Z 905.15,A -85,B 0,C 180,E1 -19465.825,E2 -19465.825} C_VEL
LIN {X 0,Y 241.969,Z 905.157,A -85,B 0,C 180,E1 -19469.588,E2 -19469.588} C_VEL
LIN {X 0,Y 241.979,Z 905.154,A -85,B 0,C 180,E1 -19473.492,E2 -19473.492} C_VEL
LIN {X 0,Y 241.98,Z 905.156,A -85,B 0,C 180,E1 -19477.583,E2 -19477.583} C_VEL
LIN {X 0,Y 241.917,Z 905.163,A -85,B 0,C 180,E1 -19481.926,E2 -19481.926} C_VEL
LIN {X 0,Y 241.908,Z 905.163,A -85,B 0,C 180,E1 -19486.577,E2 -19486.577} C_VEL
LIN {X 0,Y 241.914,Z 905.161,A -85,B 0,C 180,E1 -19489.752,E2 -19489.752} C_VEL
LIN {X 0,Y 241.282,Z 905.244,A -85,B 0,C 180,E1 -19491.142,E2 -19491.142} C_VEL
LIN {X 0,Y 238.446,Z 905.601,A -85,B 0,C 180,E1 -19493.409,E2 -19493.409} C_VEL
LIN {X 0,Y 236.031,Z 905.9,A -85,B 0,C 180,E1 -19495.257,E2 -19495.257} C_VEL
LIN {X 0,Y 235.015,Z 906.024,A -85,B 0,C 180,E1 -19496.69,E2 -19496.69} C_VEL
LIN {X 0,Y 234.944,Z 906.03,A -85,B 0,C 180,E1 -19497.176,E2 -19497.176} C_VEL
LIN {X 0,Y 235.16,Z 906.143,A -85,B 0,C 180,E1 -19501.834,E2 -19501.834} C_VEL
LIN {X 0,Y 236.774,Z 914.458,A -85,B 0,C 180,E1 -19505.445,E2 -19505.445} C_VEL
LIN {X 0,Y 236.412,Z 918.794,A -85,B 0,C 180,E1 -19507.265,E2 -19507.265} C_VEL
LIN {X 0,Y 235.652,Z 924.193,A -85,B 0,C 180,E1 -19509.429,E2 -19509.429} C_VEL
LIN {X 0,Y 236.359,Z 941.018,A -85,B 0,C 180,E1 -19510.287,E2 -19510.287} C_VEL
LIN {X 0,Y 238.497,Z 965.14,A -85,B 0,C 180,E1 -19511.515,E2 -19511.515} C_VEL
LIN {X 0,Y 237.341,Z 1003.885,A -85,B 0,C 180,E1 -19513.495,E2 -19513.495} C_VEL
LIN {X 0,Y 236.55,Z 1016.217,A -85,B 0,C 180,E1 -19514.49,E2 -19514.49} C_VEL
LIN {X 0,Y 236.038,Z 1025.955,A -85,B 0,C 180,E1 -19515.56,E2 -19515.56} C_VEL
LIN {X 0,Y 235.311,Z 1036.611,A -85,B 0,C 180,E1 -19517.055,E2 -19517.055} C_VEL
LIN {X 0,Y 234.674,Z 1045.977,A -85,B 0,C 180,E1 -19518.775,E2 -19518.775} C_VEL
LIN {X 0,Y 234.148,Z 1053.575,A -85,B 0,C 180,E1 -19520.498,E2 -19520.498} C_VEL
LIN {X 0,Y 233.812,Z 1059.886,A -85,B 0,C 180,E1 -19522.227,E2 -19522.227} C_VEL
LIN {X 0,Y 233.602,Z 1064.846,A -85,B 0,C 180,E1 -19523.857,E2 -19523.857} C_VEL
LIN {X 0,Y 233.417,Z 1069.437,A -85,B 0,C 180,E1 -19525.683,E2 -19525.683} C_VEL
LIN {X 0,Y 233.259,Z 1072.971,A -85,B 0,C 180,E1 -19527.409,E2 -19527.409} C_VEL
LIN {X 0,Y 233.158,Z 1076.974,A -85,B 0,C 180,E1 -19530,E2 -19530} C_VEL
LIN {X 0,Y 232.948,Z 1078.807,A -85,B 0,C 180,E1 -19531.729,E2 -19531.729} C_VEL
LIN {X 0,Y 232.951,Z 1080.139,A -85,B 0,C 180,E1 -19533.459,E2 -19533.459} C_VEL
LIN {X 0,Y 232.878,Z 1080.934,A -85,B 0,C 180,E1 -19535.194,E2 -19535.194} C_VEL
LIN {X 0,Y 233.074,Z 1081.135,A -85,B 0,C 180,E1 -19536.927,E2 -19536.927} C_VEL
LIN {X 0,Y 233.467,Z 1080.854,A -85,B 0,C 180,E1 -19538.656,E2 -19538.656} C_VEL
LIN {X 0,Y 234.116,Z 1080.128,A -85,B 0,C 180,E1 -19540.376,E2 -19540.376} C_VEL
LIN {X 0,Y 234.999,Z 1078.917,A -85,B 0,C 180,E1 -19542.084,E2 -19542.084} C_VEL
LIN {X 0,Y 236.769,Z 1076.017,A -85,B 0,C 180,E1 -19544.614,E2 -19544.614} C_VEL
LIN {X 0,Y 239.03,Z 1071.891,A -85,B 0,C 180,E1 -19547.099,E2 -19547.099} C_VEL
LIN {X 0,Y 241.855,Z 1066.44,A -85,B 0,C 180,E1 -19549.522,E2 -19549.522} C_VEL
LIN {X 0,Y 245.277,Z 1059.424,A -85,B 0,C 180,E1 -19551.869,E2 -19551.869} C_VEL
LIN {X 0,Y 248.569,Z 1052.054,A -85,B 0,C 180,E1 -19553.759,E2 -19553.759} C_VEL
LIN {X 0,Y 251.471,Z 1044.952,A -85,B 0,C 180,E1 -19555.226,E2 -19555.226} C_VEL
LIN {X 0,Y 254.231,Z 1037.552,A -85,B 0,C 180,E1 -19556.472,E2 -19556.472} C_VEL
LIN {X 0,Y 257.75,Z 1027.445,A -85,B 0,C 180,E1 -19557.836,E2 -19557.836} C_VEL
LIN {X 0,Y 261.083,Z 1016.161,A -85,B 0,C 180,E1 -19558.982,E2 -19558.982} C_VEL
LIN {X 0,Y 263.513,Z 1005.818,A -85,B 0,C 180,E1 -19559.784,E2 -19559.784} C_VEL
LIN {X 0,Y 265.929,Z 992.463,A -85,B 0,C 180,E1 -19560.555,E2 -19560.555} C_VEL
LIN {X 0,Y 268.527,Z 974.459,A -85,B 0,C 180,E1 -19561.474,E2 -19561.474} C_VEL
LIN {X 0,Y 268.096,Z 965.049,A -85,B 0,C 180,E1 -19562.624,E2 -19562.624} C_VEL
LIN {X 0,Y 266.001,Z 958.855,A -85,B 0,C 180,E1 -19564.256,E2 -19564.256} C_VEL
LIN {X 0,Y 264.038,Z 954.029,A -85,B 0,C 180,E1 -19565.92,E2 -19565.92} C_VEL
LIN {X 0,Y 262.16,Z 949.558,A -85,B 0,C 180,E1 -19567.853,E2 -19567.853} C_VEL
LIN {X 0,Y 259.617,Z 944.026,A -85,B 0,C 180,E1 -19571.719,E2 -19571.719} C_VEL
LIN {X 0,Y 259.303,Z 943.101,A -85,B 0,C 180,E1 -19572.655,E2 -19572.655} C_VEL
LIN {X 0,Y 258.858,Z 942.036,A -85,B 0,C 180,E1 -19575.099,E2 -19575.099} C_VEL
LIN {X 0,Y 259.372,Z 941.858,A -85,B 0,C 180,E1 -19577.824,E2 -19577.824} C_VEL
LIN {X 0,Y 261.54,Z 944.823,A -85,B 0,C 180,E1 -19581.711,E2 -19581.711} C_VEL
LIN {X 0,Y 262.383,Z 945.913,A -85,B 0,C 180,E1 -19582.6,E2 -19582.6} C_VEL
LIN {X 0,Y 264.615,Z 949.472,A -85,B 0,C 180,E1 -19584.703,E2 -19584.703} C_VEL
LIN {X 0,Y 266.929,Z 953.62,A -85,B 0,C 180,E1 -19586.493,E2 -19586.493} C_VEL
LIN {X 0,Y 269.394,Z 958.661,A -85,B 0,C 180,E1 -19588.16,E2 -19588.16} C_VEL
LIN {X 0,Y 270.127,Z 960.291,A -85,B 0,C 180,E1 -19588.607,E2 -19588.607} C_VEL
LIN {X 0,Y 265.401,Z 990.521,A -85,B 0,C 180,E1 -19590.176,E2 -19590.176} C_VEL
LIN {X 0,Y 263.09,Z 1001.767,A -85,B 0,C 180,E1 -19591.042,E2 -19591.042} C_VEL
LIN {X 0,Y 260.59,Z 1011.713,A -85,B 0,C 180,E1 -19592.057,E2 -19592.057} C_VEL
LIN {X 0,Y 257.35,Z 1022.317,A -85,B 0,C 180,E1 -19593.437,E2 -19593.437} C_VEL
LIN {X 0,Y 253.96,Z 1031.602,A -85,B 0,C 180,E1 -19595.038,E2 -19595.038} C_VEL
LIN {X 0,Y 251.201,Z 1038.474,A -85,B 0,C 180,E1 -19596.505,E2 -19596.505} C_VEL
LIN {X 0,Y 247.989,Z 1045.555,A -85,B 0,C 180,E1 -19598.383,E2 -19598.383} C_VEL
LIN {X 0,Y 244.551,Z 1052.251,A -85,B 0,C 180,E1 -19600.702,E2 -19600.702} C_VEL
LIN {X 0,Y 242.477,Z 1055.869,A -85,B 0,C 180,E1 -19602.283,E2 -19602.283} C_VEL
LIN {X 0,Y 239.65,Z 1059.979,A -85,B 0,C 180,E1 -19604.697,E2 -19604.697} C_VEL
LIN {X 0,Y 238.11,Z 1062.055,A -85,B 0,C 180,E1 -19606.343,E2 -19606.343} C_VEL
LIN {X 0,Y 236.845,Z 1063.556,A -85,B 0,C 180,E1 -19608.012,E2 -19608.012} C_VEL
LIN {X 0,Y 235.793,Z 1064.476,A -85,B 0,C 180,E1 -19609.699,E2 -19609.699} C_VEL
LIN {X 0,Y 234.824,Z 1064.932,A -85,B 0,C 180,E1 -19611.394,E2 -19611.394} C_VEL
LIN {X 0,Y 233.997,Z 1064.923,A -85,B 0,C 180,E1 -19613.101,E2 -19613.101} C_VEL
LIN {X 0,Y 233.49,Z 1064.395,A -85,B 0,C 180,E1 -19614.82,E2 -19614.82} C_VEL
LIN {X 0,Y 233.181,Z 1063.264,A -85,B 0,C 180,E1 -19616.545,E2 -19616.545} C_VEL
LIN {X 0,Y 232.924,Z 1060.683,A -85,B 0,C 180,E1 -19619.136,E2 -19619.136} C_VEL
LIN {X 0,Y 232.926,Z 1056.736,A -85,B 0,C 180,E1 -19621.73,E2 -19621.73} C_VEL
LIN {X 0,Y 233.015,Z 1052.338,A -85,B 0,C 180,E1 -19623.892,E2 -19623.892} C_VEL
LIN {X 0,Y 233.224,Z 1046.74,A -85,B 0,C 180,E1 -19626.054,E2 -19626.054} C_VEL
LIN {X 0,Y 233.697,Z 1039.796,A -85,B 0,C 180,E1 -19628.213,E2 -19628.213} C_VEL
LIN {X 0,Y 234.291,Z 1031.074,A -85,B 0,C 180,E1 -19630.37,E2 -19630.37} C_VEL
LIN {X 0,Y 234.921,Z 1022.305,A -85,B 0,C 180,E1 -19632.089,E2 -19632.089} C_VEL
LIN {X 0,Y 235.615,Z 1012.922,A -85,B 0,C 180,E1 -19633.586,E2 -19633.586} C_VEL
LIN {X 0,Y 236.418,Z 1000.865,A -85,B 0,C 180,E1 -19635.078,E2 -19635.078} C_VEL
LIN {X 0,Y 236.953,Z 990.392,A -85,B 0,C 180,E1 -19636.035,E2 -19636.035} C_VEL
LIN {X 0,Y 237.351,Z 979.984,A -85,B 0,C 180,E1 -19636.726,E2 -19636.726} C_VEL
LIN {X 0,Y 238.974,Z 931.611,A -85,B 0,C 180,E1 -19639.098,E2 -19639.098} C_VEL
LIN {X 0,Y 235.67,Z 908.34,A -85,B 0,C 180,E1 -19640.321,E2 -19640.321} C_VEL
LIN {X 0,Y 235.226,Z 905.983,A -85,B 0,C 180,E1 -19640.467,E2 -19640.467} C_VEL
LIN {X 0,Y 234.942,Z 906.029,A -85,B 0,C 180,E1 -19646.18,E2 -19646.18} C_VEL
LIN {X 0,Y 234.9,Z 906.032,A -85,B 0,C 180,E1 -19650.573,E2 -19650.573} C_VEL
LIN {X 0,Y 234.924,Z 906.032,A -85,B 0,C 180,E1 -19654.64,E2 -19654.64} C_VEL
LIN {X 0,Y 234.914,Z 906.03,A -85,B 0,C 180,E1 -19658.936,E2 -19658.936} C_VEL
LIN {X 0,Y 234.854,Z 906.042,A -85,B 0,C 180,E1 -19663.495,E2 -19663.495} C_VEL
LIN {X 0,Y 234.863,Z 906.039,A -85,B 0,C 180,E1 -19666.509,E2 -19666.509} C_VEL
LIN {X 0,Y 234.92,Z 906.032,A -85,B 0,C 180,E1 -19671.079,E2 -19671.079} C_VEL
LIN {X 0,Y 234.928,Z 906.03,A -85,B 0,C 180,E1 -19675.362,E2 -19675.362} C_VEL
LIN {X 0,Y 234.902,Z 906.033,A -85,B 0,C 180,E1 -19679.428,E2 -19679.428} C_VEL
LIN {X 0,Y 234.972,Z 906.025,A -85,B 0,C 180,E1 -19683.807,E2 -19683.807} C_VEL
LIN {X 0,Y 234.969,Z 906.024,A -85,B 0,C 180,E1 -19688.008,E2 -19688.008} C_VEL
LIN {X 0,Y 235.059,Z 906.018,A -85,B 0,C 180,E1 -19693.094,E2 -19693.094} C_VEL
LIN {X 0,Y 235.1,Z 906.01,A -85,B 0,C 180,E1 -19697.922,E2 -19697.922} C_VEL
LIN {X 0,Y 235.323,Z 905.985,A -85,B 0,C 180,E1 -19701.412,E2 -19701.412} C_VEL
LIN {X 0,Y 235.356,Z 905.978,A -85,B 0,C 180,E1 -19703.14,E2 -19703.14} C_VEL
LIN {X 0,Y 235.568,Z 905.953,A -85,B 0,C 180,E1 -19708.291,E2 -19708.291} C_VEL
LIN {X 0,Y 235.568,Z 905.953,A -85,B 0,C 180,E1 -19711.71,E2 -19711.71} C_VEL
LIN {X 0,Y 235.355,Z 905.978,A -85,B 0,C 180,E1 -19716.86,E2 -19716.86} C_VEL
LIN {X 0,Y 235.213,Z 905.999,A -85,B 0,C 180,E1 -19720.328,E2 -19720.328} C_VEL
LIN {X 0,Y 235.046,Z 906.015,A -85,B 0,C 180,E1 -19725.611,E2 -19725.611} C_VEL
LIN {X 0,Y 234.962,Z 906.029,A -85,B 0,C 180,E1 -19729.21,E2 -19729.21} C_VEL
LIN {X 0,Y 234.913,Z 906.034,A -85,B 0,C 180,E1 -19732.888,E2 -19732.888} C_VEL
LIN {X 0,Y 234.93,Z 906.032,A -85,B 0,C 180,E1 -19736.663,E2 -19736.663} C_VEL
LIN {X 0,Y 234.903,Z 906.033,A -85,B 0,C 180,E1 -19740.572,E2 -19740.572} C_VEL
LIN {X 0,Y 234.929,Z 906.03,A -85,B 0,C 180,E1 -19744.639,E2 -19744.639} C_VEL
LIN {X 0,Y 234.916,Z 906.032,A -85,B 0,C 180,E1 -19748.935,E2 -19748.935} C_VEL
LIN {X 0,Y 234.865,Z 906.039,A -85,B 0,C 180,E1 -19753.492,E2 -19753.492} C_VEL
LIN {X 0,Y 234.865,Z 906.04,A -85,B 0,C 180,E1 -19756.508,E2 -19756.508} C_VEL
LIN {X 0,Y 234.922,Z 906.029,A -85,B 0,C 180,E1 -19761.078,E2 -19761.078} C_VEL
LIN {X 0,Y 234.927,Z 906.031,A -85,B 0,C 180,E1 -19765.36,E2 -19765.36} C_VEL
LIN {X 0,Y 234.903,Z 906.031,A -85,B 0,C 180,E1 -19769.427,E2 -19769.427} C_VEL
LIN {X 0,Y 234.944,Z 906.029,A -85,B 0,C 180,E1 -19773.82,E2 -19773.82} C_VEL
LIN {X 0,Y 234.938,Z 906.031,A -85,B 0,C 180,E1 -19778.962,E2 -19778.962} C_VEL
LIN {X 0,Y 235.053,Z 906.019,A -85,B 0,C 180,E1 -19783.097,E2 -19783.097} C_VEL
LIN {X 0,Y 235.088,Z 906.009,A -85,B 0,C 180,E1 -19787.92,E2 -19787.92} C_VEL
LIN {X 0,Y 235.318,Z 905.985,A -85,B 0,C 180,E1 -19791.411,E2 -19791.411} C_VEL
LIN {X 0,Y 235.354,Z 905.979,A -85,B 0,C 180,E1 -19793.139,E2 -19793.139} C_VEL
LIN {X 0,Y 235.566,Z 905.952,A -85,B 0,C 180,E1 -19798.29,E2 -19798.29} C_VEL
LIN {X 0,Y 235.565,Z 905.953,A -85,B 0,C 180,E1 -19801.709,E2 -19801.709} C_VEL
LIN {X 0,Y 235.348,Z 905.977,A -85,B 0,C 180,E1 -19806.86,E2 -19806.86} C_VEL
LIN {X 0,Y 235.21,Z 905.999,A -85,B 0,C 180,E1 -19810.327,E2 -19810.327} C_VEL
LIN {X 0,Y 235.043,Z 906.014,A -85,B 0,C 180,E1 -19815.61,E2 -19815.61} C_VEL
LIN {X 0,Y 234.958,Z 906.029,A -85,B 0,C 180,E1 -19819.209,E2 -19819.209} C_VEL
LIN {X 0,Y 234.909,Z 906.037,A -85,B 0,C 180,E1 -19822.887,E2 -19822.887} C_VEL
LIN {X 0,Y 234.926,Z 906.03,A -85,B 0,C 180,E1 -19826.662,E2 -19826.662} C_VEL
LIN {X 0,Y 234.899,Z 906.035,A -85,B 0,C 180,E1 -19830.572,E2 -19830.572} C_VEL
LIN {X 0,Y 234.925,Z 906.028,A -85,B 0,C 180,E1 -19834.638,E2 -19834.638} C_VEL
LIN {X 0,Y 234.912,Z 906.033,A -85,B 0,C 180,E1 -19838.934,E2 -19838.934} C_VEL
LIN {X 0,Y 234.86,Z 906.039,A -85,B 0,C 180,E1 -19843.491,E2 -19843.491} C_VEL
LIN {X 0,Y 234.86,Z 906.041,A -85,B 0,C 180,E1 -19846.507,E2 -19846.507} C_VEL
LIN {X 0,Y 234.917,Z 906.031,A -85,B 0,C 180,E1 -19851.078,E2 -19851.078} C_VEL
LIN {X 0,Y 234.924,Z 906.031,A -85,B 0,C 180,E1 -19855.36,E2 -19855.36} C_VEL
LIN {X 0,Y 234.944,Z 906.03,A -85,B 0,C 180,E1 -19857.176,E2 -19857.176} C_VEL
LIN {X 0,Y 234.267,Z 906.179,A -85,B 0,C 180,E1 -19858.161,E2 -19858.161} C_VEL
LIN {X 0,Y 231.39,Z 906.471,A -85,B 0,C 180,E1 -19859.715,E2 -19859.715} C_VEL
LIN {X 0,Y 228.703,Z 906.804,A -85,B 0,C 180,E1 -19861.246,E2 -19861.246} C_VEL
LIN {X 0,Y 228.21,Z 907.304,A -85,B 0,C 180,E1 -19862.02,E2 -19862.02} C_VEL
LIN {X 0,Y 228.234,Z 907.569,A -85,B 0,C 180,E1 -19862.163,E2 -19862.163} C_VEL
LIN {X 0,Y 229.728,Z 915.275,A -85,B 0,C 180,E1 -19865.606,E2 -19865.606} C_VEL
LIN {X 0,Y 228.651,Z 923.283,A -85,B 0,C 180,E1 -19869.064,E2 -19869.064} C_VEL
LIN {X 0,Y 228.584,Z 923.678,A -85,B 0,C 180,E1 -19869.234,E2 -19869.234} C_VEL
LIN {X 0,Y 229.267,Z 941.093,A -85,B 0,C 180,E1 -19870.155,E2 -19870.155} C_VEL
LIN {X 0,Y 231.39,Z 965.45,A -85,B 0,C 180,E1 -19871.449,E2 -19871.449} C_VEL
LIN {X 0,Y 230.26,Z 1003.448,A -85,B 0,C 180,E1 -19873.486,E2 -19873.486} C_VEL
LIN {X 0,Y 229.445,Z 1016.211,A -85,B 0,C 180,E1 -19874.567,E2 -19874.567} C_VEL
LIN {X 0,Y 229.026,Z 1024.967,A -85,B 0,C 180,E1 -19875.562,E2 -19875.562} C_VEL
LIN {X 0,Y 228.37,Z 1034.233,A -85,B 0,C 180,E1 -19876.881,E2 -19876.881} C_VEL
LIN {X 0,Y 227.707,Z 1044.172,A -85,B 0,C 180,E1 -19878.652,E2 -19878.652} C_VEL
LIN {X 0,Y 227.135,Z 1052.875,A -85,B 0,C 180,E1 -19880.651,E2 -19880.651} C_VEL
LIN {X 0,Y 226.813,Z 1058.077,A -85,B 0,C 180,E1 -19882.074,E2 -19882.074} C_VEL
LIN {X 0,Y 226.56,Z 1064.39,A -85,B 0,C 180,E1 -19884.163,E2 -19884.163} C_VEL
LIN {X 0,Y 226.433,Z 1067.92,A -85,B 0,C 180,E1 -19885.549,E2 -19885.549} C_VEL
LIN {X 0,Y 226.258,Z 1071.66,A -85,B 0,C 180,E1 -19887.329,E2 -19887.329} C_VEL
LIN {X 0,Y 226.146,Z 1075.853,A -85,B 0,C 180,E1 -19890,E2 -19890} C_VEL
LIN {X 0,Y 225.916,Z 1077.918,A -85,B 0,C 180,E1 -19891.782,E2 -19891.782} C_VEL
LIN {X 0,Y 225.886,Z 1079.418,A -85,B 0,C 180,E1 -19893.567,E2 -19893.567} C_VEL
LIN {X 0,Y 225.84,Z 1080.292,A -85,B 0,C 180,E1 -19895.357,E2 -19895.357} C_VEL
LIN {X 0,Y 226.045,Z 1080.69,A -85,B 0,C 180,E1 -19897.144,E2 -19897.144} C_VEL
LIN {X 0,Y 226.442,Z 1080.65,A -85,B 0,C 180,E1 -19898.927,E2 -19898.927} C_VEL
LIN {X 0,Y 227.135,Z 1080.114,A -85,B 0,C 180,E1 -19900.699,E2 -19900.699} C_VEL
LIN {X 0,Y 228.056,Z 1078.985,A -85,B 0,C 180,E1 -19902.457,E2 -19902.457} C_VEL
LIN {X 0,Y 229.925,Z 1076.481,A -85,B 0,C 180,E1 -19905.059,E2 -19905.059} C_VEL
LIN {X 0,Y 232.323,Z 1072.759,A -85,B 0,C 180,E1 -19907.608,E2 -19907.608} C_VEL
LIN {X 0,Y 235.268,Z 1067.641,A -85,B 0,C 180,E1 -19910.092,E2 -19910.092} C_VEL
LIN {X 0,Y 238.215,Z 1062.303,A -85,B 0,C 180,E1 -19912.096,E2 -19912.096} C_VEL
LIN {X 0,Y 241.595,Z 1055.71,A -85,B 0,C 180,E1 -19914.033,E2 -19914.033} C_VEL
LIN {X 0,Y 245.335,Z 1047.752,A -85,B 0,C 180,E1 -19915.903,E2 -19915.903} C_VEL
LIN {X 0,Y 249.033,Z 1038.92,A -85,B 0,C 180,E1 -19917.524,E2 -19917.524} C_VEL
LIN {X 0,Y 252.695,Z 1029.103,A -85,B 0,C 180,E1 -19918.897,E2 -19918.897} C_VEL
LIN {X 0,Y 256.7,Z 1016.895,A -85,B 0,C 180,E1 -19920.204,E2 -19920.204} C_VEL
LIN {X 0,Y 259.639,Z 1005.363,A -85,B 0,C 180,E1 -19921.116,E2 -19921.116} C_VEL
LIN {X 0,Y 262.15,Z 992.659,A -85,B 0,C 180,E1 -19921.858,E2 -19921.858} C_VEL
LIN {X 0,Y 264.651,Z 975.898,A -85,B 0,C 180,E1 -19922.748,E2 -19922.748} C_VEL
LIN {X 0,Y 264.469,Z 969.232,A -85,B 0,C 180,E1 -19923.634,E2 -19923.634} C_VEL
LIN {X 0,Y 262.644,Z 963.602,A -85,B 0,C 180,E1 -19925.24,E2 -19925.24} C_VEL
LIN {X 0,Y 261.338,Z 960.094,A -85,B 0,C 180,E1 -19926.488,E2 -19926.488} C_VEL
LIN {X 0,Y 259.596,Z 955.633,A -85,B 0,C 180,E1 -19928.512,E2 -19928.512} C_VEL
LIN {X 0,Y 257.587,Z 950.444,A -85,B 0,C 180,E1 -19932.239,E2 -19932.239} C_VEL
LIN {X 0,Y 257.155,Z 949.353,A -85,B 0,C 180,E1 -19933.91,E2 -19933.91} C_VEL
LIN {X 0,Y 257.022,Z 948.849,A -85,B 0,C 180,E1 -19935.311,E2 -19935.311} C_VEL
LIN {X 0,Y 257.586,Z 948.808,A -85,B 0,C 180,E1 -19937.954,E2 -19937.954} C_VEL
LIN {X 0,Y 259.666,Z 951.74,A -85,B 0,C 180,E1 -19941.711,E2 -19941.711} C_VEL
LIN {X 0,Y 262.072,Z 955.799,A -85,B 0,C 180,E1 -19944.25,E2 -19944.25} C_VEL
LIN {X 0,Y 264.373,Z 960.221,A -85,B 0,C 180,E1 -19946.175,E2 -19946.175} C_VEL
LIN {X 0,Y 266.16,Z 964.073,A -85,B 0,C 180,E1 -19947.47,E2 -19947.47} C_VEL
LIN {X 0,Y 261.742,Z 990.378,A -85,B 0,C 180,E1 -19948.845,E2 -19948.845} C_VEL
LIN {X 0,Y 259.267,Z 1001.602,A -85,B 0,C 180,E1 -19949.678,E2 -19949.678} C_VEL
LIN {X 0,Y 256.18,Z 1012.914,A -85,B 0,C 180,E1 -19950.86,E2 -19950.86} C_VEL
LIN {X 0,Y 252.291,Z 1024.348,A -85,B 0,C 180,E1 -19952.412,E2 -19952.412} C_VEL
LIN {X 0,Y 249.501,Z 1031.524,A -85,B 0,C 180,E1 -19953.664,E2 -19953.664} C_VEL
LIN {X 0,Y 246.513,Z 1038.377,A -85,B 0,C 180,E1 -19955.134,E2 -19955.134} C_VEL
LIN {X 0,Y 243.012,Z 1045.495,A -85,B 0,C 180,E1 -19957.02,E2 -19957.02} C_VEL
LIN {X 0,Y 239.239,Z 1052.335,A -85,B 0,C 180,E1 -19959.359,E2 -19959.359} C_VEL
LIN {X 0,Y 235.878,Z 1057.423,A -85,B 0,C 180,E1 -19961.77,E2 -19961.77} C_VEL
LIN {X 0,Y 232.916,Z 1061.24,A -85,B 0,C 180,E1 -19964.243,E2 -19964.243} C_VEL
LIN {X 0,Y 231.302,Z 1063.052,A -85,B 0,C 180,E1 -19965.933,E2 -19965.933} C_VEL
LIN {X 0,Y 229.975,Z 1064.362,A -85,B 0,C 180,E1 -19967.649,E2 -19967.649} C_VEL
LIN {X 0,Y 228.853,Z 1065.158,A -85,B 0,C 180,E1 -19969.383,E2 -19969.383} C_VEL
LIN {X 0,Y 227.819,Z 1065.384,A -85,B 0,C 180,E1 -19971.128,E2 -19971.128} C_VEL
LIN {X 0,Y 226.962,Z 1065.128,A -85,B 0,C 180,E1 -19972.886,E2 -19972.886} C_VEL
LIN {X 0,Y 226.421,Z 1064.4,A -85,B 0,C 180,E1 -19974.658,E2 -19974.658} C_VEL
LIN {X 0,Y 226.107,Z 1063.189,A -85,B 0,C 180,E1 -19976.437,E2 -19976.437} C_VEL
LIN {X 0,Y 225.857,Z 1060.245,A -85,B 0,C 180,E1 -19979.109,E2 -19979.109} C_VEL
LIN {X 0,Y 225.864,Z 1055.99,A -85,B 0,C 180,E1 -19981.784,E2 -19981.784} C_VEL
LIN {X 0,Y 225.973,Z 1050.83,A -85,B 0,C 180,E1 -19984.23,E2 -19984.23} C_VEL
LIN {X 0,Y 226.251,Z 1044.371,A -85,B 0,C 180,E1 -19986.634,E2 -19986.634} C_VEL
LIN {X 0,Y 226.782,Z 1036.465,A -85,B 0,C 180,E1 -19988.915,E2 -19988.915} C_VEL
LIN {X 0,Y 227.342,Z 1028.87,A -85,B 0,C 180,E1 -19990.69,E2 -19990.69} C_VEL
LIN {X 0,Y 228.025,Z 1019.646,A -85,B 0,C 180,E1 -19992.46,E2 -19992.46} C_VEL
LIN {X 0,Y 228.745,Z 1009.467,A -85,B 0,C 180,E1 -19994.003,E2 -19994.003} C_VEL
LIN {X 0,Y 229.4,Z 999.2,A -85,B 0,C 180,E1 -19995.209,E2 -19995.209} C_VEL
LIN {X 0,Y 229.889,Z 989.59,A -85,B 0,C 180,E1 -19996.085,E2 -19996.085} C_VEL
LIN {X 0,Y 230.386,Z 977.075,A -85,B 0,C 180,E1 -19996.904,E2 -19996.904} C_VEL
LIN {X 0,Y 231.804,Z 931.466,A -85,B 0,C 180,E1 -19999.253,E2 -19999.253} C_VEL
LIN {X 0,Y 228.661,Z 909.177,A -85,B 0,C 180,E1 -20000.46,E2 -20000.46} C_VEL
LIN {X 0,Y 228.159,Z 906.863,A -85,B 0,C 180,E1 -20000.618,E2 -20000.618} C_VEL
LIN {X 0,Y 227.904,Z 906.907,A -85,B 0,C 180,E1 -20006.583,E2 -20006.583} C_VEL
LIN {X 0,Y 227.875,Z 906.906,A -85,B 0,C 180,E1 -20010.281,E2 -20010.281} C_VEL
LIN {X 0,Y 227.877,Z 906.912,A -85,B 0,C 180,E1 -20013.722,E2 -20013.722} C_VEL
LIN {X 0,Y 227.839,Z 906.913,A -85,B 0,C 180,E1 -20018.093,E2 -20018.093} C_VEL
LIN {X 0,Y 227.786,Z 906.921,A -85,B 0,C 180,E1 -20022.75,E2 -20022.75} C_VEL
LIN {X 0,Y 227.794,Z 906.918,A -85,B 0,C 180,E1 -20027.254,E2 -20027.254} C_VEL
LIN {X 0,Y 227.842,Z 906.915,A -85,B 0,C 180,E1 -20031.909,E2 -20031.909} C_VEL
LIN {X 0,Y 227.882,Z 906.911,A -85,B 0,C 180,E1 -20036.378,E2 -20036.378} C_VEL
LIN {X 0,Y 227.88,Z 906.911,A -85,B 0,C 180,E1 -20040.432,E2 -20040.432} C_VEL
LIN {X 0,Y 227.905,Z 906.907,A -85,B 0,C 180,E1 -20044.423,E2 -20044.423} C_VEL
LIN {X 0,Y 227.929,Z 906.901,A -85,B 0,C 180,E1 -20048.284,E2 -20048.284} C_VEL
LIN {X 0,Y 228.022,Z 906.891,A -85,B 0,C 180,E1 -20053.896,E2 -20053.896} C_VEL
LIN {X 0,Y 228.058,Z 906.889,A -85,B 0,C 180,E1 -20057.543,E2 -20057.543} C_VEL
LIN {X 0,Y 228.262,Z 906.863,A -85,B 0,C 180,E1 -20061.145,E2 -20061.145} C_VEL
LIN {X 0,Y 228.309,Z 906.855,A -85,B 0,C 180,E1 -20062.927,E2 -20062.927} C_VEL
LIN {X 0,Y 228.502,Z 906.834,A -85,B 0,C 180,E1 -20068.238,E2 -20068.238} C_VEL
LIN {X 0,Y 228.501,Z 906.834,A -85,B 0,C 180,E1 -20071.763,E2 -20071.763} C_VEL
LIN {X 0,Y 228.308,Z 906.856,A -85,B 0,C 180,E1 -20077.073,E2 -20077.073} C_VEL
LIN {X 0,Y 228.143,Z 906.879,A -85,B 0,C 180,E1 -20080.652,E2 -20080.652} C_VEL
LIN {X 0,Y 228.004,Z 906.893,A -85,B 0,C 180,E1 -20086.106,E2 -20086.106} C_VEL
LIN {X 0,Y 227.923,Z 906.902,A -85,B 0,C 180,E1 -20091.717,E2 -20091.717} C_VEL
LIN {X 0,Y 227.907,Z 906.906,A -85,B 0,C 180,E1 -20096.582,E2 -20096.582} C_VEL
LIN {X 0,Y 227.878,Z 906.908,A -85,B 0,C 180,E1 -20100.28,E2 -20100.28} C_VEL
LIN {X 0,Y 227.881,Z 906.911,A -85,B 0,C 180,E1 -20103.72,E2 -20103.72} C_VEL
LIN {X 0,Y 227.844,Z 906.915,A -85,B 0,C 180,E1 -20108.092,E2 -20108.092} C_VEL
LIN {X 0,Y 227.796,Z 906.918,A -85,B 0,C 180,E1 -20112.746,E2 -20112.746} C_VEL
LIN {X 0,Y 227.796,Z 906.92,A -85,B 0,C 180,E1 -20117.253,E2 -20117.253} C_VEL
LIN {X 0,Y 227.844,Z 906.912,A -85,B 0,C 180,E1 -20121.908,E2 -20121.908} C_VEL
LIN {X 0,Y 227.882,Z 906.913,A -85,B 0,C 180,E1 -20126.377,E2 -20126.377} C_VEL
LIN {X 0,Y 227.879,Z 906.908,A -85,B 0,C 180,E1 -20130.431,E2 -20130.431} C_VEL
LIN {X 0,Y 227.87,Z 906.912,A -85,B 0,C 180,E1 -20134.418,E2 -20134.418} C_VEL
LIN {X 0,Y 227.922,Z 906.902,A -85,B 0,C 180,E1 -20138.282,E2 -20138.282} C_VEL
LIN {X 0,Y 228.003,Z 906.895,A -85,B 0,C 180,E1 -20143.893,E2 -20143.893} C_VEL
LIN {X 0,Y 228.128,Z 906.877,A -85,B 0,C 180,E1 -20149.347,E2 -20149.347} C_VEL
LIN {X 0,Y 228.306,Z 906.856,A -85,B 0,C 180,E1 -20152.926,E2 -20152.926} C_VEL
LIN {X 0,Y 228.5,Z 906.832,A -85,B 0,C 180,E1 -20158.237,E2 -20158.237} C_VEL
LIN {X 0,Y 228.499,Z 906.834,A -85,B 0,C 180,E1 -20161.762,E2 -20161.762} C_VEL
LIN {X 0,Y 228.3,Z 906.854,A -85,B 0,C 180,E1 -20167.072,E2 -20167.072} C_VEL
LIN {X 0,Y 228.14,Z 906.88,A -85,B 0,C 180,E1 -20170.651,E2 -20170.651} C_VEL
LIN {X 0,Y 228.001,Z 906.892,A -85,B 0,C 180,E1 -20176.105,E2 -20176.105} C_VEL
LIN {X 0,Y 227.92,Z 906.904,A -85,B 0,C 180,E1 -20181.716,E2 -20181.716} C_VEL
LIN {X 0,Y 227.904,Z 906.904,A -85,B 0,C 180,E1 -20186.581,E2 -20186.581} C_VEL
LIN {X 0,Y 227.874,Z 906.91,A -85,B 0,C 180,E1 -20190.28,E2 -20190.28} C_VEL
LIN {X 0,Y 227.877,Z 906.909,A -85,B 0,C 180,E1 -20193.72,E2 -20193.72} C_VEL
LIN {X 0,Y 227.839,Z 906.916,A -85,B 0,C 180,E1 -20198.091,E2 -20198.091} C_VEL
LIN {X 0,Y 227.792,Z 906.918,A -85,B 0,C 180,E1 -20202.746,E2 -20202.746} C_VEL
LIN {X 0,Y 227.791,Z 906.92,A -85,B 0,C 180,E1 -20207.252,E2 -20207.252} C_VEL
LIN {X 0,Y 227.838,Z 906.915,A -85,B 0,C 180,E1 -20211.907,E2 -20211.907} C_VEL
LIN {X 0,Y 227.878,Z 906.912,A -85,B 0,C 180,E1 -20216.377,E2 -20216.377} C_VEL
LIN {X 0,Y 228.133,Z 907.025,A -85,B 0,C 180,E1 -20221.916,E2 -20221.916} C_VEL
LIN {X 0,Y 228.234,Z 907.569,A -85,B 0,C 180,E1 -20222.163,E2 -20222.163} C_VEL
LIN {X 0,Y 228.049,Z 910.497,A -85,B 0,C 180,E1 -20223.455,E2 -20223.455} C_VEL
LIN {X 0,Y 226.885,Z 913.454,A -85,B 0,C 180,E1 -20224.725,E2 -20224.725} C_VEL
LIN {X 0,Y 221.55,Z 923.301,A -85,B 0,C 180,E1 -20229.02,E2 -20229.02} C_VEL
LIN {X 0,Y 221.963,Z 938.427,A -85,B 0,C 180,E1 -20229.906,E2 -20229.906} C_VEL
LIN {X 0,Y 224.32,Z 964.945,A -85,B 0,C 180,E1 -20231.376,E2 -20231.376} C_VEL
LIN {X 0,Y 223.167,Z 1003.38,A -85,B 0,C 180,E1 -20233.535,E2 -20233.535} C_VEL
LIN {X 0,Y 222.368,Z 1016.036,A -85,B 0,C 180,E1 -20234.651,E2 -20234.651} C_VEL
LIN {X 0,Y 221.88,Z 1025.594,A -85,B 0,C 180,E1 -20235.789,E2 -20235.789} C_VEL
LIN {X 0,Y 221.167,Z 1036.118,A -85,B 0,C 180,E1 -20237.381,E2 -20237.381} C_VEL
LIN {X 0,Y 220.547,Z 1045.443,A -85,B 0,C 180,E1 -20239.209,E2 -20239.209} C_VEL
LIN {X 0,Y 220.106,Z 1052.138,A -85,B 0,C 180,E1 -20240.813,E2 -20240.813} C_VEL
LIN {X 0,Y 219.76,Z 1058.508,A -85,B 0,C 180,E1 -20242.65,E2 -20242.65} C_VEL
LIN {X 0,Y 219.519,Z 1064.993,A -85,B 0,C 180,E1 -20244.949,E2 -20244.949} C_VEL
LIN {X 0,Y 219.281,Z 1070.101,A -85,B 0,C 180,E1 -20247.244,E2 -20247.244} C_VEL
LIN {X 0,Y 219.132,Z 1074.721,A -85,B 0,C 180,E1 -20250,E2 -20250} C_VEL
LIN {X 0,Y 218.905,Z 1076.931,A -85,B 0,C 180,E1 -20251.839,E2 -20251.839} C_VEL
LIN {X 0,Y 218.844,Z 1078.507,A -85,B 0,C 180,E1 -20253.682,E2 -20253.682} C_VEL
LIN {X 0,Y 218.794,Z 1079.592,A -85,B 0,C 180,E1 -20255.53,E2 -20255.53} C_VEL
LIN {X 0,Y 219.008,Z 1080.238,A -85,B 0,C 180,E1 -20257.375,E2 -20257.375} C_VEL
LIN {X 0,Y 219.417,Z 1080.368,A -85,B 0,C 180,E1 -20259.215,E2 -20259.215} C_VEL
LIN {X 0,Y 220.171,Z 1079.929,A -85,B 0,C 180,E1 -20261.041,E2 -20261.041} C_VEL
LIN {X 0,Y 221.131,Z 1079.057,A -85,B 0,C 180,E1 -20262.854,E2 -20262.854} C_VEL
LIN {X 0,Y 222.356,Z 1077.741,A -85,B 0,C 180,E1 -20264.646,E2 -20264.646} C_VEL
LIN {X 0,Y 224.72,Z 1074.701,A -85,B 0,C 180,E1 -20267.284,E2 -20267.284} C_VEL
LIN {X 0,Y 227.602,Z 1070.51,A -85,B 0,C 180,E1 -20269.856,E2 -20269.856} C_VEL
LIN {X 0,Y 231.176,Z 1064.942,A -85,B 0,C 180,E1 -20272.334,E2 -20272.334} C_VEL
LIN {X 0,Y 235.321,Z 1057.845,A -85,B 0,C 180,E1 -20274.716,E2 -20274.716} C_VEL
LIN {X 0,Y 239.148,Z 1050.406,A -85,B 0,C 180,E1 -20276.626,E2 -20276.626} C_VEL
LIN {X 0,Y 243.458,Z 1041.287,A -85,B 0,C 180,E1 -20278.445,E2 -20278.445} C_VEL
LIN {X 0,Y 247.77,Z 1031.105,A -85,B 0,C 180,E1 -20279.995,E2 -20279.995} C_VEL
LIN {X 0,Y 251.396,Z 1021.083,A -85,B 0,C 180,E1 -20281.143,E2 -20281.143} C_VEL
LIN {X 0,Y 255.171,Z 1008.566,A -85,B 0,C 180,E1 -20282.251,E2 -20282.251} C_VEL
LIN {X 0,Y 257.931,Z 996.519,A -85,B 0,C 180,E1 -20283.021,E2 -20283.021} C_VEL
LIN {X 0,Y 261.082,Z 978.002,A -85,B 0,C 180,E1 -20284.018,E2 -20284.018} C_VEL
LIN {X 0,Y 261.019,Z 973.555,A -85,B 0,C 180,E1 -20284.624,E2 -20284.624} C_VEL
LIN {X 0,Y 259.277,Z 967.769,A -85,B 0,C 180,E1 -20286.444,E2 -20286.444} C_VEL
LIN {X 0,Y 258.313,Z 965.076,A -85,B 0,C 180,E1 -20287.565,E2 -20287.565} C_VEL
LIN {X 0,Y 257.302,Z 962.099,A -85,B 0,C 180,E1 -20288.919,E2 -20288.919} C_VEL
LIN {X 0,Y 255.565,Z 956.786,A -85,B 0,C 180,E1 -20292.802,E2 -20292.802} C_VEL
LIN {X 0,Y 255.228,Z 955.655,A -85,B 0,C 180,E1 -20295.72,E2 -20295.72} C_VEL
LIN {X 0,Y 255.833,Z 955.917,A -85,B 0,C 180,E1 -20298.263,E2 -20298.263} C_VEL
LIN {X 0,Y 257.853,Z 958.934,A -85,B 0,C 180,E1 -20301.845,E2 -20301.845} C_VEL
LIN {X 0,Y 259.697,Z 962.405,A -85,B 0,C 180,E1 -20303.931,E2 -20303.931} C_VEL
LIN {X 0,Y 261.759,Z 966.603,A -85,B 0,C 180,E1 -20305.769,E2 -20305.769} C_VEL
LIN {X 0,Y 262.352,Z 968.094,A -85,B 0,C 180,E1 -20306.277,E2 -20306.277} C_VEL
LIN {X 0,Y 258.235,Z 990.999,A -85,B 0,C 180,E1 -20307.487,E2 -20307.487} C_VEL
LIN {X 0,Y 255.684,Z 1001.728,A -85,B 0,C 180,E1 -20308.286,E2 -20308.286} C_VEL
LIN {X 0,Y 252.387,Z 1012.978,A -85,B 0,C 180,E1 -20309.457,E2 -20309.457} C_VEL
LIN {X 0,Y 248.712,Z 1023.394,A -85,B 0,C 180,E1 -20310.828,E2 -20310.828} C_VEL
LIN {X 0,Y 245.252,Z 1031.595,A -85,B 0,C 180,E1 -20312.248,E2 -20312.248} C_VEL
LIN {X 0,Y 241.24,Z 1040.018,A -85,B 0,C 180,E1 -20314.089,E2 -20314.089} C_VEL
LIN {X 0,Y 237.527,Z 1046.931,A -85,B 0,C 180,E1 -20315.994,E2 -20315.994} C_VEL
LIN {X 0,Y 234.104,Z 1052.466,A -85,B 0,C 180,E1 -20317.96,E2 -20317.96} C_VEL
LIN {X 0,Y 230.459,Z 1057.624,A -85,B 0,C 180,E1 -20320.401,E2 -20320.401} C_VEL
LIN {X 0,Y 227.18,Z 1061.458,A -85,B 0,C 180,E1 -20322.91,E2 -20322.91} C_VEL
LIN {X 0,Y 224.502,Z 1064.049,A -85,B 0,C 180,E1 -20325.497,E2 -20325.497} C_VEL
LIN {X 0,Y 223.085,Z 1065.098,A -85,B 0,C 180,E1 -20327.261,E2 -20327.261} C_VEL
LIN {X 0,Y 221.91,Z 1065.686,A -85,B 0,C 180,E1 -20329.047,E2 -20329.047} C_VEL
LIN {X 0,Y 220.818,Z 1065.804,A -85,B 0,C 180,E1 -20330.844,E2 -20330.844} C_VEL
LIN {X 0,Y 219.933,Z 1065.324,A -85,B 0,C 180,E1 -20332.657,E2 -20332.657} C_VEL
LIN {X 0,Y 219.358,Z 1064.349,A -85,B 0,C 180,E1 -20334.485,E2 -20334.485} C_VEL
LIN {X 0,Y 219.036,Z 1062.905,A -85,B 0,C 180,E1 -20336.322,E2 -20336.322} C_VEL
LIN {X 0,Y 218.792,Z 1059.703,A -85,B 0,C 180,E1 -20339.081,E2 -20339.081} C_VEL
LIN {X 0,Y 218.753,Z 1056.863,A -85,B 0,C 180,E1 -20340.921,E2 -20340.921} C_VEL
LIN {X 0,Y 218.876,Z 1051.315,A -85,B 0,C 180,E1 -20343.683,E2 -20343.683} C_VEL
LIN {X 0,Y 219.135,Z 1044.889,A -85,B 0,C 180,E1 -20346.166,E2 -20346.166} C_VEL
LIN {X 0,Y 219.591,Z 1037.965,A -85,B 0,C 180,E1 -20348.282,E2 -20348.282} C_VEL
LIN {X 0,Y 220.199,Z 1029.631,A -85,B 0,C 180,E1 -20350.343,E2 -20350.343} C_VEL
LIN {X 0,Y 220.852,Z 1020.577,A -85,B 0,C 180,E1 -20352.171,E2 -20352.171} C_VEL
LIN {X 0,Y 221.674,Z 1009.037,A -85,B 0,C 180,E1 -20353.99,E2 -20353.99} C_VEL
LIN {X 0,Y 222.324,Z 998.616,A -85,B 0,C 180,E1 -20355.235,E2 -20355.235} C_VEL
LIN {X 0,Y 222.847,Z 987.438,A -85,B 0,C 180,E1 -20356.255,E2 -20356.255} C_VEL
LIN {X 0,Y 223.555,Z 969.443,A -85,B 0,C 180,E1 -20357.319,E2 -20357.319} C_VEL
LIN {X 0,Y 224.756,Z 932.128,A -85,B 0,C 180,E1 -20359.319,E2 -20359.319} C_VEL
LIN {X 0,Y 221.578,Z 909.901,A -85,B 0,C 180,E1 -20360.566,E2 -20360.566} C_VEL
LIN {X 0,Y 221.134,Z 907.738,A -85,B 0,C 180,E1 -20360.711,E2 -20360.711} C_VEL
LIN {X 0,Y 220.851,Z 907.788,A -85,B 0,C 180,E1 -20366.998,E2 -20366.998} C_VEL
LIN {X 0,Y 220.82,Z 907.786,A -85,B 0,C 180,E1 -20370.76,E2 -20370.76} C_VEL
LIN {X 0,Y 220.793,Z 907.793,A -85,B 0,C 180,E1 -20374.958,E2 -20374.958} C_VEL
LIN {X 0,Y 220.798,Z 907.792,A -85,B 0,C 180,E1 -20377.274,E2 -20377.274} C_VEL
LIN {X 0,Y 220.748,Z 907.801,A -85,B 0,C 180,E1 -20381.959,E2 -20381.959} C_VEL
LIN {X 0,Y 220.757,Z 907.798,A -85,B 0,C 180,E1 -20385.542,E2 -20385.542} C_VEL
LIN {X 0,Y 220.785,Z 907.795,A -85,B 0,C 180,E1 -20390.459,E2 -20390.459} C_VEL
LIN {X 0,Y 220.828,Z 907.789,A -85,B 0,C 180,E1 -20392.794,E2 -20392.794} C_VEL
LIN {X 0,Y 220.815,Z 907.786,A -85,B 0,C 180,E1 -20397.244,E2 -20397.244} C_VEL
LIN {X 0,Y 220.807,Z 907.791,A -85,B 0,C 180,E1 -20401.483,E2 -20401.483} C_VEL
LIN {X 0,Y 220.848,Z 907.783,A -85,B 0,C 180,E1 -20405.563,E2 -20405.563} C_VEL
LIN {X 0,Y 220.857,Z 907.785,A -85,B 0,C 180,E1 -20409.511,E2 -20409.511} C_VEL
LIN {X 0,Y 220.98,Z 907.771,A -85,B 0,C 180,E1 -20413.368,E2 -20413.368} C_VEL
LIN {X 0,Y 221.066,Z 907.758,A -85,B 0,C 180,E1 -20419.004,E2 -20419.004} C_VEL
LIN {X 0,Y 221.247,Z 907.735,A -85,B 0,C 180,E1 -20422.7,E2 -20422.7} C_VEL
LIN {X 0,Y 221.439,Z 907.714,A -85,B 0,C 180,E1 -20428.182,E2 -20428.182} C_VEL
LIN {X 0,Y 221.546,Z 907.703,A -85,B 0,C 180,E1 -20430,E2 -20430} C_VEL
LIN {X 0,Y 221.439,Z 907.714,A -85,B 0,C 180,E1 -20431.819,E2 -20431.819} C_VEL
LIN {X 0,Y 221.246,Z 907.735,A -85,B 0,C 180,E1 -20437.3,E2 -20437.3} C_VEL
LIN {X 0,Y 221.063,Z 907.759,A -85,B 0,C 180,E1 -20440.997,E2 -20440.997} C_VEL
LIN {X 0,Y 220.97,Z 907.772,A -85,B 0,C 180,E1 -20446.634,E2 -20446.634} C_VEL
LIN {X 0,Y 220.85,Z 907.786,A -85,B 0,C 180,E1 -20450.491,E2 -20450.491} C_VEL
LIN {X 0,Y 220.801,Z 907.789,A -85,B 0,C 180,E1 -20454.443,E2 -20454.443} C_VEL
LIN {X 0,Y 220.804,Z 907.791,A -85,B 0,C 180,E1 -20458.519,E2 -20458.519} C_VEL
LIN {X 0,Y 220.817,Z 907.785,A -85,B 0,C 180,E1 -20462.757,E2 -20462.757} C_VEL
LIN {X 0,Y 220.805,Z 907.792,A -85,B 0,C 180,E1 -20467.275,E2 -20467.275} C_VEL
LIN {X 0,Y 220.758,Z 907.797,A -85,B 0,C 180,E1 -20471.956,E2 -20471.956} C_VEL
LIN {X 0,Y 220.76,Z 907.797,A -85,B 0,C 180,E1 -20475.541,E2 -20475.541} C_VEL
LIN {X 0,Y 220.787,Z 907.792,A -85,B 0,C 180,E1 -20480.458,E2 -20480.458} C_VEL
LIN {X 0,Y 220.829,Z 907.788,A -85,B 0,C 180,E1 -20482.793,E2 -20482.793} C_VEL
LIN {X 0,Y 220.816,Z 907.789,A -85,B 0,C 180,E1 -20487.243,E2 -20487.243} C_VEL
LIN {X 0,Y 220.803,Z 907.789,A -85,B 0,C 180,E1 -20491.481,E2 -20491.481} C_VEL
LIN {X 0,Y 220.8,Z 907.792,A -85,B 0,C 180,E1 -20495.556,E2 -20495.556} C_VEL
LIN {X 0,Y 220.849,Z 907.784,A -85,B 0,C 180,E1 -20499.509,E2 -20499.509} C_VEL
LIN {X 0,Y 220.969,Z 907.774,A -85,B 0,C 180,E1 -20503.366,E2 -20503.366} C_VEL
LIN {X 0,Y 221.053,Z 907.756,A -85,B 0,C 180,E1 -20509.002,E2 -20509.002} C_VEL
LIN {X 0,Y 221.244,Z 907.736,A -85,B 0,C 180,E1 -20512.699,E2 -20512.699} C_VEL
LIN {X 0,Y 221.437,Z 907.712,A -85,B 0,C 180,E1 -20518.18,E2 -20518.18} C_VEL
LIN {X 0,Y 221.544,Z 907.701,A -85,B 0,C 180,E1 -20519.999,E2 -20519.999} C_VEL
LIN {X 0,Y 221.436,Z 907.714,A -85,B 0,C 180,E1 -20521.818,E2 -20521.818} C_VEL
LIN {X 0,Y 221.237,Z 907.733,A -85,B 0,C 180,E1 -20527.299,E2 -20527.299} C_VEL
LIN {X 0,Y 221.06,Z 907.76,A -85,B 0,C 180,E1 -20530.996,E2 -20530.996} C_VEL
LIN {X 0,Y 220.967,Z 907.77,A -85,B 0,C 180,E1 -20536.633,E2 -20536.633} C_VEL
LIN {X 0,Y 220.847,Z 907.787,A -85,B 0,C 180,E1 -20540.49,E2 -20540.49} C_VEL
LIN {X 0,Y 220.797,Z 907.79,A -85,B 0,C 180,E1 -20544.442,E2 -20544.442} C_VEL
LIN {X 0,Y 220.8,Z 907.791,A -85,B 0,C 180,E1 -20548.518,E2 -20548.518} C_VEL
LIN {X 0,Y 220.812,Z 907.789,A -85,B 0,C 180,E1 -20552.756,E2 -20552.756} C_VEL
LIN {X 0,Y 220.801,Z 907.792,A -85,B 0,C 180,E1 -20557.274,E2 -20557.274} C_VEL
LIN {X 0,Y 220.754,Z 907.798,A -85,B 0,C 180,E1 -20561.955,E2 -20561.955} C_VEL
LIN {X 0,Y 220.755,Z 907.796,A -85,B 0,C 180,E1 -20565.541,E2 -20565.541} C_VEL
LIN {X 0,Y 220.782,Z 907.795,A -85,B 0,C 180,E1 -20570.457,E2 -20570.457} C_VEL
LIN {X 0,Y 220.824,Z 907.786,A -85,B 0,C 180,E1 -20572.792,E2 -20572.792} C_VEL
LIN {X 0,Y 220.819,Z 907.789,A -85,B 0,C 180,E1 -20577.244,E2 -20577.244} C_VEL
LIN {X 0,Y 221.113,Z 907.91,A -85,B 0,C 180,E1 -20582.025,E2 -20582.025} C_VEL
LIN {X 0,Y 222.628,Z 916.034,A -85,B 0,C 180,E1 -20585.77,E2 -20585.77} C_VEL
LIN {X 0,Y 221.55,Z 923.301,A -85,B 0,C 180,E1 -20589.02,E2 -20589.02} C_VEL
LIN {X 0,Y 216.351,Z 931.032,A -85,B 0,C 180,E1 -20589.391,E2 -20589.391} C_VEL
LIN {X 0,Y 214.352,Z 936.834,A -85,B 0,C 180,E1 -20589.705,E2 -20589.705} C_VEL
LIN {X 0,Y 214.09,Z 940.852,A -85,B 0,C 180,E1 -20589.835,E2 -20589.835} C_VEL
LIN {X 0,Y 216.154,Z 953.59,A -85,B 0,C 180,E1 -20590.69,E2 -20590.69} C_VEL
LIN {X 0,Y 217.21,Z 965.425,A -85,B 0,C 180,E1 -20591.366,E2 -20591.366} C_VEL
LIN {X 0,Y 216.07,Z 1003.306,A -85,B 0,C 180,E1 -20593.586,E2 -20593.586} C_VEL
LIN {X 0,Y 215.29,Z 1015.77,A -85,B 0,C 180,E1 -20594.74,E2 -20594.74} C_VEL
LIN {X 0,Y 214.886,Z 1024.394,A -85,B 0,C 180,E1 -20595.8,E2 -20595.8} C_VEL
LIN {X 0,Y 214.227,Z 1033.535,A -85,B 0,C 180,E1 -20597.206,E2 -20597.206} C_VEL
LIN {X 0,Y 213.597,Z 1043.404,A -85,B 0,C 180,E1 -20599.094,E2 -20599.094} C_VEL
LIN {X 0,Y 213.103,Z 1051.379,A -85,B 0,C 180,E1 -20601.035,E2 -20601.035} C_VEL
LIN {X 0,Y 212.765,Z 1058.612,A -85,B 0,C 180,E1 -20603.195,E2 -20603.195} C_VEL
LIN {X 0,Y 212.538,Z 1064.241,A -85,B 0,C 180,E1 -20605.258,E2 -20605.258} C_VEL
LIN {X 0,Y 212.326,Z 1068.461,A -85,B 0,C 180,E1 -20607.154,E2 -20607.154} C_VEL
LIN {X 0,Y 212.182,Z 1071.892,A -85,B 0,C 180,E1 -20609.051,E2 -20609.051} C_VEL
LIN {X 0,Y 212.011,Z 1074.645,A -85,B 0,C 180,E1 -20610.949,E2 -20610.949} C_VEL
LIN {X 0,Y 211.821,Z 1077.557,A -85,B 0,C 180,E1 -20613.804,E2 -20613.804} C_VEL
LIN {X 0,Y 211.758,Z 1078.891,A -85,B 0,C 180,E1 -20615.714,E2 -20615.714} C_VEL
LIN {X 0,Y 211.992,Z 1079.674,A -85,B 0,C 180,E1 -20617.62,E2 -20617.62} C_VEL
LIN {X 0,Y 212.413,Z 1079.911,A -85,B 0,C 180,E1 -20619.522,E2 -20619.522} C_VEL
LIN {X 0,Y 213.191,Z 1079.738,A -85,B 0,C 180,E1 -20621.408,E2 -20621.408} C_VEL
LIN {X 0,Y 214.224,Z 1079.127,A -85,B 0,C 180,E1 -20623.276,E2 -20623.276} C_VEL
LIN {X 0,Y 215.506,Z 1077.958,A -85,B 0,C 180,E1 -20625.123,E2 -20625.123} C_VEL
LIN {X 0,Y 217.989,Z 1075.352,A -85,B 0,C 180,E1 -20627.835,E2 -20627.835} C_VEL
LIN {X 0,Y 221.011,Z 1071.51,A -85,B 0,C 180,E1 -20630.474,E2 -20630.474} C_VEL
LIN {X 0,Y 224.746,Z 1066.379,A -85,B 0,C 180,E1 -20633.009,E2 -20633.009} C_VEL
LIN {X 0,Y 228.288,Z 1060.991,A -85,B 0,C 180,E1 -20635.043,E2 -20635.043} C_VEL
LIN {X 0,Y 233.052,Z 1053.039,A -85,B 0,C 180,E1 -20637.379,E2 -20637.379} C_VEL
LIN {X 0,Y 237.472,Z 1044.714,A -85,B 0,C 180,E1 -20639.23,E2 -20639.23} C_VEL
LIN {X 0,Y 241.92,Z 1035.324,A -85,B 0,C 180,E1 -20640.798,E2 -20640.798} C_VEL
LIN {X 0,Y 246.169,Z 1025.313,A -85,B 0,C 180,E1 -20642.122,E2 -20642.122} C_VEL
LIN {X 0,Y 250.069,Z 1014.125,A -85,B 0,C 180,E1 -20643.232,E2 -20643.232} C_VEL
LIN {X 0,Y 253.112,Z 1003.39,A -85,B 0,C 180,E1 -20644.037,E2 -20644.037} C_VEL
LIN {X 0,Y 256.741,Z 986.147,A -85,B 0,C 180,E1 -20645.001,E2 -20645.001} C_VEL
LIN {X 0,Y 257.798,Z 979.827,A -85,B 0,C 180,E1 -20645.384,E2 -20645.384} C_VEL
LIN {X 0,Y 257.752,Z 977.934,A -85,B 0,C 180,E1 -20645.696,E2 -20645.696} C_VEL
LIN {X 0,Y 256.332,Z 972.557,A -85,B 0,C 180,E1 -20647.502,E2 -20647.502} C_VEL
LIN {X 0,Y 254.978,Z 968.371,A -85,B 0,C 180,E1 -20649.488,E2 -20649.488} C_VEL
LIN {X 0,Y 253.606,Z 963.57,A -85,B 0,C 180,E1 -20653.049,E2 -20653.049} C_VEL
LIN {X 0,Y 253.353,Z 962.641,A -85,B 0,C 180,E1 -20655.116,E2 -20655.116} C_VEL
LIN {X 0,Y 253.878,Z 962.597,A -85,B 0,C 180,E1 -20657.96,E2 -20657.96} C_VEL
LIN {X 0,Y 255.656,Z 965.423,A -85,B 0,C 180,E1 -20661.432,E2 -20661.432} C_VEL
LIN {X 0,Y 257.249,Z 968.719,A -85,B 0,C 180,E1 -20663.436,E2 -20663.436} C_VEL
LIN {X 0,Y 258.845,Z 972.18,A -85,B 0,C 180,E1 -20665.022,E2 -20665.022} C_VEL
LIN {X 0,Y 254.977,Z 991.9,A -85,B 0,C 180,E1 -20666.093,E2 -20666.093} C_VEL
LIN {X 0,Y 251.812,Z 1003.994,A -85,B 0,C 180,E1 -20667.028,E2 -20667.028} C_VEL
LIN {X 0,Y 248.737,Z 1013.746,A -85,B 0,C 180,E1 -20668.058,E2 -20668.058} C_VEL
LIN {X 0,Y 244.928,Z 1023.704,A -85,B 0,C 180,E1 -20669.382,E2 -20669.382} C_VEL
LIN {X 0,Y 240.317,Z 1033.704,A -85,B 0,C 180,E1 -20671.15,E2 -20671.15} C_VEL
LIN {X 0,Y 236.9,Z 1040.307,A -85,B 0,C 180,E1 -20672.625,E2 -20672.625} C_VEL
LIN {X 0,Y 232.924,Z 1047.12,A -85,B 0,C 180,E1 -20674.536,E2 -20674.536} C_VEL
LIN {X 0,Y 229.169,Z 1052.743,A -85,B 0,C 180,E1 -20676.505,E2 -20676.505} C_VEL
LIN {X 0,Y 225.196,Z 1057.895,A -85,B 0,C 180,E1 -20678.968,E2 -20678.968} C_VEL
LIN {X 0,Y 221.605,Z 1061.729,A -85,B 0,C 180,E1 -20681.511,E2 -20681.511} C_VEL
LIN {X 0,Y 219.515,Z 1063.642,A -85,B 0,C 180,E1 -20683.254,E2 -20683.254} C_VEL
LIN {X 0,Y 217.712,Z 1065.042,A -85,B 0,C 180,E1 -20685.035,E2 -20685.035} C_VEL
LIN {X 0,Y 216.222,Z 1065.841,A -85,B 0,C 180,E1 -20686.849,E2 -20686.849} C_VEL
LIN {X 0,Y 214.701,Z 1066.184,A -85,B 0,C 180,E1 -20689.117,E2 -20689.117} C_VEL
LIN {X 0,Y 212.894,Z 1065.438,A -85,B 0,C 180,E1 -20692.413,E2 -20692.413} C_VEL
LIN {X 0,Y 212.299,Z 1064.277,A -85,B 0,C 180,E1 -20694.301,E2 -20694.301} C_VEL
LIN {X 0,Y 211.854,Z 1061.631,A -85,B 0,C 180,E1 -20697.149,E2 -20697.149} C_VEL
LIN {X 0,Y 211.699,Z 1057.641,A -85,B 0,C 180,E1 -20700.001,E2 -20700.001} C_VEL
LIN {X 0,Y 211.771,Z 1053.267,A -85,B 0,C 180,E1 -20702.378,E2 -20702.378} C_VEL
LIN {X 0,Y 211.878,Z 1048.79,A -85,B 0,C 180,E1 -20704.356,E2 -20704.356} C_VEL
LIN {X 0,Y 212.199,Z 1042.389,A -85,B 0,C 180,E1 -20706.657,E2 -20706.657} C_VEL
LIN {X 0,Y 212.652,Z 1035.945,A -85,B 0,C 180,E1 -20708.554,E2 -20708.554} C_VEL
LIN {X 0,Y 213.267,Z 1027.174,A -85,B 0,C 180,E1 -20710.683,E2 -20710.683} C_VEL
LIN {X 0,Y 213.987,Z 1017.369,A -85,B 0,C 180,E1 -20712.568,E2 -20712.568} C_VEL
LIN {X 0,Y 214.624,Z 1008.212,A -85,B 0,C 180,E1 -20713.976,E2 -20713.976} C_VEL
LIN {X 0,Y 215.283,Z 997.699,A -85,B 0,C 180,E1 -20715.261,E2 -20715.261} C_VEL
LIN {X 0,Y 215.789,Z 986.14,A -85,B 0,C 180,E1 -20716.315,E2 -20716.315} C_VEL
LIN {X 0,Y 216.835,Z 958.979,A -85,B 0,C 180,E1 -20717.934,E2 -20717.934} C_VEL
LIN {X 0,Y 217.629,Z 932.512,A -85,B 0,C 180,E1 -20719.406,E2 -20719.406} C_VEL
LIN {X 0,Y 214.627,Z 911.332,A -85,B 0,C 180,E1 -20720.647,E2 -20720.647} C_VEL
LIN {X 0,Y 214.064,Z 908.618,A -85,B 0,C 180,E1 -20720.871,E2 -20720.871} C_VEL
LIN {X 0,Y 213.771,Z 908.67,A -85,B 0,C 180,E1 -20725.303,E2 -20725.303} C_VEL
LIN {X 0,Y 213.75,Z 908.668,A -85,B 0,C 180,E1 -20729.552,E2 -20729.552} C_VEL
LIN {X 0,Y 213.755,Z 908.67,A -85,B 0,C 180,E1 -20733.984,E2 -20733.984} C_VEL
LIN {X 0,Y 213.703,Z 908.672,A -85,B 0,C 180,E1 -20738.672,E2 -20738.672} C_VEL
LIN {X 0,Y 213.703,Z 908.678,A -85,B 0,C 180,E1 -20743.655,E2 -20743.655} C_VEL
LIN {X 0,Y 213.704,Z 908.675,A -85,B 0,C 180,E1 -20746.346,E2 -20746.346} C_VEL
LIN {X 0,Y 213.708,Z 908.671,A -85,B 0,C 180,E1 -20749.148,E2 -20749.148} C_VEL
LIN {X 0,Y 213.744,Z 908.671,A -85,B 0,C 180,E1 -20753.712,E2 -20753.712} C_VEL
LIN {X 0,Y 213.762,Z 908.666,A -85,B 0,C 180,E1 -20758.262,E2 -20758.262} C_VEL
LIN {X 0,Y 213.792,Z 908.667,A -85,B 0,C 180,E1 -20762.599,E2 -20762.599} C_VEL
LIN {X 0,Y 213.804,Z 908.662,A -85,B 0,C 180,E1 -20766.987,E2 -20766.987} C_VEL
LIN {X 0,Y 213.889,Z 908.654,A -85,B 0,C 180,E1 -20772.799,E2 -20772.799} C_VEL
LIN {X 0,Y 213.936,Z 908.643,A -85,B 0,C 180,E1 -20776.706,E2 -20776.706} C_VEL
LIN {X 0,Y 214.14,Z 908.621,A -85,B 0,C 180,E1 -20780.555,E2 -20780.555} C_VEL
LIN {X 0,Y 214.072,Z 908.627,A -85,B 0,C 180,E1 -20784.348,E2 -20784.348} C_VEL
LIN {X 0,Y 214.379,Z 908.594,A -85,B 0,C 180,E1 -20788.122,E2 -20788.122} C_VEL
LIN {X 0,Y 214.514,Z 908.579,A -85,B 0,C 180,E1 -20790,E2 -20790} C_VEL
LIN {X 0,Y 214.077,Z 908.628,A -85,B 0,C 180,E1 -20793.765,E2 -20793.765} C_VEL
LIN {X 0,Y 214.187,Z 908.615,A -85,B 0,C 180,E1 -20797.542,E2 -20797.542} C_VEL
LIN {X 0,Y 213.992,Z 908.638,A -85,B 0,C 180,E1 -20801.365,E2 -20801.365} C_VEL
LIN {X 0,Y 213.872,Z 908.654,A -85,B 0,C 180,E1 -20805.242,E2 -20805.242} C_VEL
LIN {X 0,Y 213.794,Z 908.666,A -85,B 0,C 180,E1 -20809.192,E2 -20809.192} C_VEL
LIN {X 0,Y 213.769,Z 908.667,A -85,B 0,C 180,E1 -20813.237,E2 -20813.237} C_VEL
LIN {X 0,Y 213.789,Z 908.667,A -85,B 0,C 180,E1 -20817.426,E2 -20817.426} C_VEL
LIN {X 0,Y 213.763,Z 908.665,A -85,B 0,C 180,E1 -20821.739,E2 -20821.739} C_VEL
LIN {X 0,Y 213.746,Z 908.671,A -85,B 0,C 180,E1 -20826.289,E2 -20826.289} C_VEL
LIN {X 0,Y 213.705,Z 908.672,A -85,B 0,C 180,E1 -20831.128,E2 -20831.128} C_VEL
LIN {X 0,Y 213.706,Z 908.675,A -85,B 0,C 180,E1 -20833.679,E2 -20833.679} C_VEL
LIN {X 0,Y 213.706,Z 908.677,A -85,B 0,C 180,E1 -20836.345,E2 -20836.345} C_VEL
LIN {X 0,Y 213.709,Z 908.673,A -85,B 0,C 180,E1 -20839.146,E2 -20839.146} C_VEL
LIN {X 0,Y 213.745,Z 908.67,A -85,B 0,C 180,E1 -20843.711,E2 -20843.711} C_VEL
LIN {X 0,Y 213.763,Z 908.669,A -85,B 0,C 180,E1 -20848.26,E2 -20848.26} C_VEL
LIN {X 0,Y 213.787,Z 908.666,A -85,B 0,C 180,E1 -20852.597,E2 -20852.597} C_VEL
LIN {X 0,Y 213.783,Z 908.667,A -85,B 0,C 180,E1 -20856.999,E2 -20856.999} C_VEL
LIN {X 0,Y 213.881,Z 908.654,A -85,B 0,C 180,E1 -20862.797,E2 -20862.797} C_VEL
LIN {X 0,Y 213.915,Z 908.648,A -85,B 0,C 180,E1 -20866.703,E2 -20866.703} C_VEL
LIN {X 0,Y 214.137,Z 908.62,A -85,B 0,C 180,E1 -20870.554,E2 -20870.554} C_VEL
LIN {X 0,Y 214.07,Z 908.63,A -85,B 0,C 180,E1 -20874.347,E2 -20874.347} C_VEL
LIN {X 0,Y 214.377,Z 908.591,A -85,B 0,C 180,E1 -20878.12,E2 -20878.12} C_VEL
LIN {X 0,Y 214.512,Z 908.577,A -85,B 0,C 180,E1 -20879.999,E2 -20879.999} C_VEL
LIN {X 0,Y 214.075,Z 908.63,A -85,B 0,C 180,E1 -20883.764,E2 -20883.764} C_VEL
LIN {X 0,Y 214.179,Z 908.612,A -85,B 0,C 180,E1 -20887.541,E2 -20887.541} C_VEL
LIN {X 0,Y 213.989,Z 908.64,A -85,B 0,C 180,E1 -20891.364,E2 -20891.364} C_VEL
LIN {X 0,Y 213.868,Z 908.652,A -85,B 0,C 180,E1 -20895.241,E2 -20895.241} C_VEL
LIN {X 0,Y 213.791,Z 908.666,A -85,B 0,C 180,E1 -20899.191,E2 -20899.191} C_VEL
LIN {X 0,Y 213.765,Z 908.668,A -85,B 0,C 180,E1 -20903.236,E2 -20903.236} C_VEL
LIN {X 0,Y 213.785,Z 908.667,A -85,B 0,C 180,E1 -20907.426,E2 -20907.426} C_VEL
LIN {X 0,Y 213.759,Z 908.669,A -85,B 0,C 180,E1 -20911.738,E2 -20911.738} C_VEL
LIN {X 0,Y 213.741,Z 908.67,A -85,B 0,C 180,E1 -20916.288,E2 -20916.288} C_VEL
LIN {X 0,Y 213.7,Z 908.676,A -85,B 0,C 180,E1 -20921.127,E2 -20921.127} C_VEL
LIN {X 0,Y 213.701,Z 908.675,A -85,B 0,C 180,E1 -20923.679,E2 -20923.679} C_VEL
LIN {X 0,Y 213.701,Z 908.678,A -85,B 0,C 180,E1 -20926.345,E2 -20926.345} C_VEL
LIN {X 0,Y 213.705,Z 908.675,A -85,B 0,C 180,E1 -20929.146,E2 -20929.146} C_VEL
LIN {X 0,Y 213.74,Z 908.667,A -85,B 0,C 180,E1 -20933.71,E2 -20933.71} C_VEL
LIN {X 0,Y 213.801,Z 908.666,A -85,B 0,C 180,E1 -20938.721,E2 -20938.721} C_VEL
LIN {X 0,Y 214.049,Z 908.646,A -85,B 0,C 180,E1 -20942.096,E2 -20942.096} C_VEL
LIN {X 0,Y 215.487,Z 915.86,A -85,B 0,C 180,E1 -20945.537,E2 -20945.537} C_VEL
LIN {X 0,Y 214.651,Z 922.007,A -85,B 0,C 180,E1 -20948.386,E2 -20948.386} C_VEL
LIN {X 0,Y 214.472,Z 923.203,A -85,B 0,C 180,E1 -20948.939,E2 -20948.939} C_VEL
LIN {X 0,Y 214.905,Z 939.286,A -85,B 0,C 180,E1 -20949.864,E2 -20949.864} C_VEL
LIN {X 0,Y 216.154,Z 953.59,A -85,B 0,C 180,E1 -20950.69,E2 -20950.69} C_VEL
LIN {X 0,Y 215.811,Z 959.362,A -85,B 0,C 180,E1 -20951.012,E2 -20951.012} C_VEL
LIN {X 0,Y 213.193,Z 968.745,A -85,B 0,C 180,E1 -20951.54,E2 -20951.54} C_VEL
LIN {X 0,Y 210.345,Z 978.126,A -85,B 0,C 180,E1 -20952.105,E2 -20952.105} C_VEL
LIN {X 0,Y 209.601,Z 983.915,A -85,B 0,C 180,E1 -20952.457,E2 -20952.457} C_VEL
LIN {X 0,Y 208.93,Z 1004.104,A -85,B 0,C 180,E1 -20953.762,E2 -20953.762} C_VEL
LIN {X 0,Y 208.195,Z 1016.1,A -85,B 0,C 180,E1 -20954.959,E2 -20954.959} C_VEL
LIN {X 0,Y 207.767,Z 1024.568,A -85,B 0,C 180,E1 -20956.053,E2 -20956.053} C_VEL
LIN {X 0,Y 207.08,Z 1035.046,A -85,B 0,C 180,E1 -20957.753,E2 -20957.753} C_VEL
LIN {X 0,Y 206.515,Z 1044.418,A -85,B 0,C 180,E1 -20959.708,E2 -20959.708} C_VEL
LIN {X 0,Y 206.037,Z 1052.158,A -85,B 0,C 180,E1 -20961.714,E2 -20961.714} C_VEL
LIN {X 0,Y 205.769,Z 1057.729,A -85,B 0,C 180,E1 -20963.448,E2 -20963.448} C_VEL
LIN {X 0,Y 205.556,Z 1063.397,A -85,B 0,C 180,E1 -20965.588,E2 -20965.588} C_VEL
LIN {X 0,Y 205.309,Z 1068.582,A -85,B 0,C 180,E1 -20968.038,E2 -20968.038} C_VEL
LIN {X 0,Y 205.178,Z 1071.883,A -85,B 0,C 180,E1 -20970,E2 -20970} C_VEL
LIN {X 0,Y 204.951,Z 1074.521,A -85,B 0,C 180,E1 -20971.965,E2 -20971.965} C_VEL
LIN {X 0,Y 204.795,Z 1076.587,A -85,B 0,C 180,E1 -20973.935,E2 -20973.935} C_VEL
LIN {X 0,Y 204.753,Z 1078.005,A -85,B 0,C 180,E1 -20975.91,E2 -20975.91} C_VEL
LIN {X 0,Y 204.992,Z 1078.937,A -85,B 0,C 180,E1 -20977.882,E2 -20977.882} C_VEL
LIN {X 0,Y 205.425,Z 1079.447,A -85,B 0,C 180,E1 -20979.849,E2 -20979.849} C_VEL
LIN {X 0,Y 206.231,Z 1079.524,A -85,B 0,C 180,E1 -20981.798,E2 -20981.798} C_VEL
LIN {X 0,Y 207.319,Z 1079.022,A -85,B 0,C 180,E1 -20983.727,E2 -20983.727} C_VEL
LIN {X 0,Y 208.677,Z 1078.074,A -85,B 0,C 180,E1 -20985.63,E2 -20985.63} C_VEL
LIN {X 0,Y 210.346,Z 1076.695,A -85,B 0,C 180,E1 -20987.5,E2 -20987.5} C_VEL
LIN {X 0,Y 213.341,Z 1073.651,A -85,B 0,C 180,E1 -20990.236,E2 -20990.236} C_VEL
LIN {X 0,Y 216.966,Z 1069.429,A -85,B 0,C 180,E1 -20992.874,E2 -20992.874} C_VEL
LIN {X 0,Y 221.245,Z 1063.917,A -85,B 0,C 180,E1 -20995.394,E2 -20995.394} C_VEL
LIN {X 0,Y 226.132,Z 1056.863,A -85,B 0,C 180,E1 -20997.787,E2 -20997.787} C_VEL
LIN {X 0,Y 231.547,Z 1047.85,A -85,B 0,C 180,E1 -21000.054,E2 -21000.054} C_VEL
LIN {X 0,Y 236.703,Z 1038.511,A -85,B 0,C 180,E1 -21001.804,E2 -21001.804} C_VEL
LIN {X 0,Y 241.047,Z 1029.122,A -85,B 0,C 180,E1 -21003.139,E2 -21003.139} C_VEL
LIN {X 0,Y 245.104,Z 1019.171,A -85,B 0,C 180,E1 -21004.244,E2 -21004.244} C_VEL
LIN {X 0,Y 248.999,Z 1007.758,A -85,B 0,C 180,E1 -21005.23,E2 -21005.23} C_VEL
LIN {X 0,Y 252.311,Z 994.743,A -85,B 0,C 180,E1 -21006.041,E2 -21006.041} C_VEL
LIN {X 0,Y 254.68,Z 982.643,A -85,B 0,C 180,E1 -21006.709,E2 -21006.709} C_VEL
LIN {X 0,Y 253.598,Z 978.05,A -85,B 0,C 180,E1 -21008.378,E2 -21008.378} C_VEL
LIN {X 0,Y 252.705,Z 974.664,A -85,B 0,C 180,E1 -21010.032,E2 -21010.032} C_VEL
LIN {X 0,Y 251.662,Z 970.199,A -85,B 0,C 180,E1 -21013.442,E2 -21013.442} C_VEL
LIN {X 0,Y 251.517,Z 969.39,A -85,B 0,C 180,E1 -21015.689,E2 -21015.689} C_VEL
LIN {X 0,Y 251.997,Z 969.557,A -85,B 0,C 180,E1 -21017.985,E2 -21017.985} C_VEL
LIN {X 0,Y 253.537,Z 972.103,A -85,B 0,C 180,E1 -21021.133,E2 -21021.133} C_VEL
LIN {X 0,Y 254.943,Z 975.281,A -85,B 0,C 180,E1 -21023.077,E2 -21023.077} C_VEL
LIN {X 0,Y 255.464,Z 976.887,A -85,B 0,C 180,E1 -21023.778,E2 -21023.778} C_VEL
LIN {X 0,Y 251.816,Z 994.026,A -85,B 0,C 180,E1 -21024.718,E2 -21024.718} C_VEL
LIN {X 0,Y 248.686,Z 1004.957,A -85,B 0,C 180,E1 -21025.584,E2 -21025.584} C_VEL
LIN {X 0,Y 245.004,Z 1015.583,A -85,B 0,C 180,E1 -21026.729,E2 -21026.729} C_VEL
LIN {X 0,Y 240.323,Z 1026.429,A -85,B 0,C 180,E1 -21028.239,E2 -21028.239} C_VEL
LIN {X 0,Y 236.436,Z 1034.237,A -85,B 0,C 180,E1 -21029.648,E2 -21029.648} C_VEL
LIN {X 0,Y 231.992,Z 1042.069,A -85,B 0,C 180,E1 -21031.453,E2 -21031.453} C_VEL
LIN {X 0,Y 226.85,Z 1049.87,A -85,B 0,C 180,E1 -21033.803,E2 -21033.803} C_VEL
LIN {X 0,Y 222.936,Z 1054.924,A -85,B 0,C 180,E1 -21035.807,E2 -21035.807} C_VEL
LIN {X 0,Y 218.782,Z 1059.652,A -85,B 0,C 180,E1 -21038.321,E2 -21038.321} C_VEL
LIN {X 0,Y 215.014,Z 1063.15,A -85,B 0,C 180,E1 -21040.922,E2 -21040.922} C_VEL
LIN {X 0,Y 212.819,Z 1064.717,A -85,B 0,C 180,E1 -21042.711,E2 -21042.711} C_VEL
LIN {X 0,Y 210.913,Z 1065.829,A -85,B 0,C 180,E1 -21044.54,E2 -21044.54} C_VEL
LIN {X 0,Y 209.343,Z 1066.494,A -85,B 0,C 180,E1 -21046.409,E2 -21046.409} C_VEL
LIN {X 0,Y 208.044,Z 1066.621,A -85,B 0,C 180,E1 -21048.307,E2 -21048.307} C_VEL
LIN {X 0,Y 206.857,Z 1066.21,A -85,B 0,C 180,E1 -21050.22,E2 -21050.22} C_VEL
LIN {X 0,Y 205.868,Z 1065.359,A -85,B 0,C 180,E1 -21052.152,E2 -21052.152} C_VEL
LIN {X 0,Y 205.244,Z 1064.048,A -85,B 0,C 180,E1 -21054.105,E2 -21054.105} C_VEL
LIN {X 0,Y 204.802,Z 1061.026,A -85,B 0,C 180,E1 -21057.05,E2 -21057.05} C_VEL
LIN {X 0,Y 204.64,Z 1056.772,A -85,B 0,C 180,E1 -21060.001,E2 -21060.001} C_VEL
LIN {X 0,Y 204.745,Z 1052.103,A -85,B 0,C 180,E1 -21062.46,E2 -21062.46} C_VEL
LIN {X 0,Y 204.896,Z 1046.156,A -85,B 0,C 180,E1 -21064.962,E2 -21064.962} C_VEL
LIN {X 0,Y 205.397,Z 1038.34,A -85,B 0,C 180,E1 -21067.564,E2 -21067.564} C_VEL
LIN {X 0,Y 205.982,Z 1029.819,A -85,B 0,C 180,E1 -21069.824,E2 -21069.824} C_VEL
LIN {X 0,Y 206.638,Z 1020.757,A -85,B 0,C 180,E1 -21071.776,E2 -21071.776} C_VEL
LIN {X 0,Y 207.342,Z 1010.783,A -85,B 0,C 180,E1 -21073.477,E2 -21073.477} C_VEL
LIN {X 0,Y 208.111,Z 999.785,A -85,B 0,C 180,E1 -21074.923,E2 -21074.923} C_VEL
LIN {X 0,Y 208.669,Z 987.604,A -85,B 0,C 180,E1 -21076.134,E2 -21076.134} C_VEL
LIN {X 0,Y 209.519,Z 965.987,A -85,B 0,C 180,E1 -21077.509,E2 -21077.509} C_VEL
LIN {X 0,Y 210.491,Z 932.53,A -85,B 0,C 180,E1 -21079.49,E2 -21079.49} C_VEL
LIN {X 0,Y 207.732,Z 912.966,A -85,B 0,C 180,E1 -21080.667,E2 -21080.667} C_VEL
LIN {X 0,Y 207.023,Z 909.495,A -85,B 0,C 180,E1 -21080.902,E2 -21080.902} C_VEL
LIN {X 0,Y 206.698,Z 909.548,A -85,B 0,C 180,E1 -21086.234,E2 -21086.234} C_VEL
LIN {X 0,Y 206.696,Z 909.544,A -85,B 0,C 180,E1 -21090.667,E2 -21090.667} C_VEL
LIN {X 0,Y 206.701,Z 909.55,A -85,B 0,C 180,E1 -21095.312,E2 -21095.312} C_VEL
LIN {X 0,Y 206.647,Z 909.554,A -85,B 0,C 180,E1 -21100.256,E2 -21100.256} C_VEL
LIN {X 0,Y 206.631,Z 909.557,A -85,B 0,C 180,E1 -21104.418,E2 -21104.418} C_VEL
LIN {X 0,Y 206.636,Z 909.554,A -85,B 0,C 180,E1 -21108.441,E2 -21108.441} C_VEL
LIN {X 0,Y 206.671,Z 909.555,A -85,B 0,C 180,E1 -21112.259,E2 -21112.259} C_VEL
LIN {X 0,Y 206.697,Z 909.544,A -85,B 0,C 180,E1 -21117.042,E2 -21117.042} C_VEL
LIN {X 0,Y 206.713,Z 909.547,A -85,B 0,C 180,E1 -21122.127,E2 -21122.127} C_VEL
LIN {X 0,Y 206.742,Z 909.541,A -85,B 0,C 180,E1 -21126.615,E2 -21126.615} C_VEL
LIN {X 0,Y 206.826,Z 909.532,A -85,B 0,C 180,E1 -21132.193,E2 -21132.193} C_VEL
LIN {X 0,Y 206.877,Z 909.521,A -85,B 0,C 180,E1 -21136.243,E2 -21136.243} C_VEL
LIN {X 0,Y 207.084,Z 909.5,A -85,B 0,C 180,E1 -21140.231,E2 -21140.231} C_VEL
LIN {X 0,Y 207.037,Z 909.504,A -85,B 0,C 180,E1 -21144.155,E2 -21144.155} C_VEL
LIN {X 0,Y 207.321,Z 909.473,A -85,B 0,C 180,E1 -21148.058,E2 -21148.058} C_VEL
LIN {X 0,Y 207.481,Z 909.455,A -85,B 0,C 180,E1 -21150,E2 -21150} C_VEL
LIN {X 0,Y 207.024,Z 909.507,A -85,B 0,C 180,E1 -21153.893,E2 -21153.893} C_VEL
LIN {X 0,Y 207.132,Z 909.494,A -85,B 0,C 180,E1 -21157.801,E2 -21157.801} C_VEL
LIN {X 0,Y 206.912,Z 909.521,A -85,B 0,C 180,E1 -21161.76,E2 -21161.76} C_VEL
LIN {X 0,Y 206.805,Z 909.533,A -85,B 0,C 180,E1 -21165.776,E2 -21165.776} C_VEL
LIN {X 0,Y 206.715,Z 909.546,A -85,B 0,C 180,E1 -21169.876,E2 -21169.876} C_VEL
LIN {X 0,Y 206.696,Z 909.545,A -85,B 0,C 180,E1 -21174.081,E2 -21174.081} C_VEL
LIN {X 0,Y 206.691,Z 909.549,A -85,B 0,C 180,E1 -21178.427,E2 -21178.427} C_VEL
LIN {X 0,Y 206.699,Z 909.544,A -85,B 0,C 180,E1 -21182.958,E2 -21182.958} C_VEL
LIN {X 0,Y 206.672,Z 909.554,A -85,B 0,C 180,E1 -21187.742,E2 -21187.742} C_VEL
LIN {X 0,Y 206.637,Z 909.554,A -85,B 0,C 180,E1 -21191.56,E2 -21191.56} C_VEL
LIN {X 0,Y 206.634,Z 909.557,A -85,B 0,C 180,E1 -21195.582,E2 -21195.582} C_VEL
LIN {X 0,Y 206.653,Z 909.553,A -85,B 0,C 180,E1 -21199.745,E2 -21199.745} C_VEL
LIN {X 0,Y 206.703,Z 909.55,A -85,B 0,C 180,E1 -21204.688,E2 -21204.688} C_VEL
LIN {X 0,Y 206.698,Z 909.544,A -85,B 0,C 180,E1 -21209.334,E2 -21209.334} C_VEL
LIN {X 0,Y 206.687,Z 909.549,A -85,B 0,C 180,E1 -21213.765,E2 -21213.765} C_VEL
LIN {X 0,Y 206.709,Z 909.544,A -85,B 0,C 180,E1 -21218.037,E2 -21218.037} C_VEL
LIN {X 0,Y 206.806,Z 909.534,A -85,B 0,C 180,E1 -21222.19,E2 -21222.19} C_VEL
LIN {X 0,Y 206.856,Z 909.527,A -85,B 0,C 180,E1 -21226.241,E2 -21226.241} C_VEL
LIN {X 0,Y 207.081,Z 909.499,A -85,B 0,C 180,E1 -21230.229,E2 -21230.229} C_VEL
LIN {X 0,Y 207.035,Z 909.507,A -85,B 0,C 180,E1 -21234.154,E2 -21234.154} C_VEL
LIN {X 0,Y 207.319,Z 909.47,A -85,B 0,C 180,E1 -21238.056,E2 -21238.056} C_VEL
LIN {X 0,Y 207.479,Z 909.452,A -85,B 0,C 180,E1 -21239.999,E2 -21239.999} C_VEL
LIN {X 0,Y 207.022,Z 909.51,A -85,B 0,C 180,E1 -21243.892,E2 -21243.892} C_VEL
LIN {X 0,Y 207.123,Z 909.492,A -85,B 0,C 180,E1 -21247.8,E2 -21247.8} C_VEL
LIN {X 0,Y 206.909,Z 909.522,A -85,B 0,C 180,E1 -21251.758,E2 -21251.758} C_VEL
LIN {X 0,Y 206.802,Z 909.531,A -85,B 0,C 180,E1 -21255.775,E2 -21255.775} C_VEL
LIN {X 0,Y 206.711,Z 909.546,A -85,B 0,C 180,E1 -21259.875,E2 -21259.875} C_VEL
LIN {X 0,Y 206.692,Z 909.546,A -85,B 0,C 180,E1 -21264.08,E2 -21264.08} C_VEL
LIN {X 0,Y 206.687,Z 909.549,A -85,B 0,C 180,E1 -21268.426,E2 -21268.426} C_VEL
LIN {X 0,Y 206.695,Z 909.548,A -85,B 0,C 180,E1 -21272.957,E2 -21272.957} C_VEL
LIN {X 0,Y 206.668,Z 909.555,A -85,B 0,C 180,E1 -21277.741,E2 -21277.741} C_VEL
LIN {X 0,Y 206.633,Z 909.558,A -85,B 0,C 180,E1 -21281.559,E2 -21281.559} C_VEL
LIN {X 0,Y 206.629,Z 909.555,A -85,B 0,C 180,E1 -21285.582,E2 -21285.582} C_VEL
LIN {X 0,Y 206.648,Z 909.555,A -85,B 0,C 180,E1 -21289.745,E2 -21289.745} C_VEL
LIN {X 0,Y 206.699,Z 909.549,A -85,B 0,C 180,E1 -21294.688,E2 -21294.688} C_VEL
LIN {X 0,Y 206.767,Z 909.539,A -85,B 0,C 180,E1 -21299.346,E2 -21299.346} C_VEL
LIN {X 0,Y 207.086,Z 909.603,A -85,B 0,C 180,E1 -21302.316,E2 -21302.316} C_VEL
LIN {X 0,Y 208.395,Z 916.236,A -85,B 0,C 180,E1 -21305.581,E2 -21305.581} C_VEL
LIN {X 0,Y 207.403,Z 922.855,A -85,B 0,C 180,E1 -21308.767,E2 -21308.767} C_VEL
LIN {X 0,Y 207.841,Z 939.857,A -85,B 0,C 180,E1 -21309.817,E2 -21309.817} C_VEL
LIN {X 0,Y 210.118,Z 965.377,A -85,B 0,C 180,E1 -21311.346,E2 -21311.346} C_VEL
LIN {X 0,Y 209.601,Z 983.915,A -85,B 0,C 180,E1 -21312.457,E2 -21312.457} C_VEL
LIN {X 0,Y 208.781,Z 989.636,A -85,B 0,C 180,E1 -21312.806,E2 -21312.806} C_VEL
LIN {X 0,Y 205.545,Z 998.758,A -85,B 0,C 180,E1 -21313.433,E2 -21313.433} C_VEL
LIN {X 0,Y 202.213,Z 1007.725,A -85,B 0,C 180,E1 -21314.218,E2 -21314.218} C_VEL
LIN {X 0,Y 201.253,Z 1013.208,A -85,B 0,C 180,E1 -21314.803,E2 -21314.803} C_VEL
LIN {X 0,Y 200.775,Z 1023.067,A -85,B 0,C 180,E1 -21316.074,E2 -21316.074} C_VEL
LIN {X 0,Y 200.174,Z 1032.287,A -85,B 0,C 180,E1 -21317.581,E2 -21317.581} C_VEL
LIN {X 0,Y 199.595,Z 1042.181,A -85,B 0,C 180,E1 -21319.603,E2 -21319.603} C_VEL
LIN {X 0,Y 199.082,Z 1050.87,A -85,B 0,C 180,E1 -21321.882,E2 -21321.882} C_VEL
LIN {X 0,Y 198.784,Z 1057.2,A -85,B 0,C 180,E1 -21323.911,E2 -21323.911} C_VEL
LIN {X 0,Y 198.59,Z 1062.465,A -85,B 0,C 180,E1 -21325.941,E2 -21325.941} C_VEL
LIN {X 0,Y 198.372,Z 1066.81,A -85,B 0,C 180,E1 -21327.969,E2 -21327.969} C_VEL
LIN {X 0,Y 198.216,Z 1070.397,A -85,B 0,C 180,E1 -21330,E2 -21330} C_VEL
LIN {X 0,Y 197.978,Z 1073.207,A -85,B 0,C 180,E1 -21332.034,E2 -21332.034} C_VEL
LIN {X 0,Y 197.722,Z 1076.625,A -85,B 0,C 180,E1 -21335.59,E2 -21335.59} C_VEL
LIN {X 0,Y 197.975,Z 1078.198,A -85,B 0,C 180,E1 -21338.163,E2 -21338.163} C_VEL
LIN {X 0,Y 198.452,Z 1078.92,A -85,B 0,C 180,E1 -21340.199,E2 -21340.199} C_VEL
LIN {X 0,Y 199.29,Z 1079.088,A -85,B 0,C 180,E1 -21342.215,E2 -21342.215} C_VEL
LIN {X 0,Y 200.417,Z 1078.845,A -85,B 0,C 180,E1 -21344.209,E2 -21344.209} C_VEL
LIN {X 0,Y 201.869,Z 1078.195,A -85,B 0,C 180,E1 -21346.171,E2 -21346.171} C_VEL
LIN {X 0,Y 203.591,Z 1077.029,A -85,B 0,C 180,E1 -21348.1,E2 -21348.1} C_VEL
LIN {X 0,Y 206.733,Z 1074.407,A -85,B 0,C 180,E1 -21350.913,E2 -21350.913} C_VEL
LIN {X 0,Y 210.549,Z 1070.612,A -85,B 0,C 180,E1 -21353.612,E2 -21353.612} C_VEL
LIN {X 0,Y 214.994,Z 1065.538,A -85,B 0,C 180,E1 -21356.187,E2 -21356.187} C_VEL
LIN {X 0,Y 219.189,Z 1060.216,A -85,B 0,C 180,E1 -21358.225,E2 -21358.225} C_VEL
LIN {X 0,Y 223.778,Z 1053.828,A -85,B 0,C 180,E1 -21360.165,E2 -21360.165} C_VEL
LIN {X 0,Y 228.772,Z 1046.018,A -85,B 0,C 180,E1 -21362,E2 -21362} C_VEL
LIN {X 0,Y 234.271,Z 1036.332,A -85,B 0,C 180,E1 -21363.71,E2 -21363.71} C_VEL
LIN {X 0,Y 238.961,Z 1026.728,A -85,B 0,C 180,E1 -21364.995,E2 -21364.995} C_VEL
LIN {X 0,Y 243.321,Z 1016.238,A -85,B 0,C 180,E1 -21366.083,E2 -21366.083} C_VEL
LIN {X 0,Y 247.404,Z 1004.176,A -85,B 0,C 180,E1 -21367.019,E2 -21367.019} C_VEL
LIN {X 0,Y 250.793,Z 991.047,A -85,B 0,C 180,E1 -21367.789,E2 -21367.789} C_VEL
LIN {X 0,Y 251.696,Z 986.647,A -85,B 0,C 180,E1 -21368.022,E2 -21368.022} C_VEL
LIN {X 0,Y 251.083,Z 983.845,A -85,B 0,C 180,E1 -21369.147,E2 -21369.147} C_VEL
LIN {X 0,Y 250.454,Z 980.968,A -85,B 0,C 180,E1 -21370.584,E2 -21370.584} C_VEL
LIN {X 0,Y 249.76,Z 977.025,A -85,B 0,C 180,E1 -21373.621,E2 -21373.621} C_VEL
LIN {X 0,Y 249.629,Z 976.287,A -85,B 0,C 180,E1 -21375.265,E2 -21375.265} C_VEL
LIN {X 0,Y 250.065,Z 976.35,A -85,B 0,C 180,E1 -21377.815,E2 -21377.815} C_VEL
LIN {X 0,Y 251.438,Z 978.867,A -85,B 0,C 180,E1 -21380.878,E2 -21380.878} C_VEL
LIN {X 0,Y 252.419,Z 981.315,A -85,B 0,C 180,E1 -21382.437,E2 -21382.437} C_VEL
LIN {X 0,Y 249.107,Z 995.575,A -85,B 0,C 180,E1 -21383.257,E2 -21383.257} C_VEL
LIN {X 0,Y 245.645,Z 1006.603,A -85,B 0,C 180,E1 -21384.148,E2 -21384.148} C_VEL
LIN {X 0,Y 241.349,Z 1017.934,A -85,B 0,C 180,E1 -21385.402,E2 -21385.402} C_VEL
LIN {X 0,Y 236.79,Z 1027.571,A -85,B 0,C 180,E1 -21386.769,E2 -21386.769} C_VEL
LIN {X 0,Y 232.814,Z 1034.9,A -85,B 0,C 180,E1 -21388.112,E2 -21388.112} C_VEL
LIN {X 0,Y 227.985,Z 1042.851,A -85,B 0,C 180,E1 -21389.939,E2 -21389.939} C_VEL
LIN {X 0,Y 223.41,Z 1049.303,A -85,B 0,C 180,E1 -21391.845,E2 -21391.845} C_VEL
LIN {X 0,Y 218.305,Z 1055.386,A -85,B 0,C 180,E1 -21394.24,E2 -21394.24} C_VEL
LIN {X 0,Y 213.766,Z 1060.095,A -85,B 0,C 180,E1 -21396.765,E2 -21396.765} C_VEL
LIN {X 0,Y 210.993,Z 1062.485,A -85,B 0,C 180,E1 -21398.507,E2 -21398.507} C_VEL
LIN {X 0,Y 208.424,Z 1064.401,A -85,B 0,C 180,E1 -21400.295,E2 -21400.295} C_VEL
LIN {X 0,Y 206.135,Z 1065.815,A -85,B 0,C 180,E1 -21402.132,E2 -21402.132} C_VEL
LIN {X 0,Y 204.138,Z 1066.625,A -85,B 0,C 180,E1 -21404.014,E2 -21404.014} C_VEL
LIN {X 0,Y 202.474,Z 1066.972,A -85,B 0,C 180,E1 -21405.939,E2 -21405.939} C_VEL
LIN {X 0,Y 201.108,Z 1066.908,A -85,B 0,C 180,E1 -21407.897,E2 -21407.897} C_VEL
LIN {X 0,Y 199.624,Z 1066.149,A -85,B 0,C 180,E1 -21410.323,E2 -21410.323} C_VEL
LIN {X 0,Y 198.194,Z 1063.667,A -85,B 0,C 180,E1 -21413.894,E2 -21413.894} C_VEL
LIN {X 0,Y 197.751,Z 1060.359,A -85,B 0,C 180,E1 -21416.945,E2 -21416.945} C_VEL
LIN {X 0,Y 197.591,Z 1055.802,A -85,B 0,C 180,E1 -21420.001,E2 -21420.001} C_VEL
LIN {X 0,Y 197.748,Z 1049.676,A -85,B 0,C 180,E1 -21423.057,E2 -21423.057} C_VEL
LIN {X 0,Y 197.999,Z 1043.062,A -85,B 0,C 180,E1 -21425.624,E2 -21425.624} C_VEL
LIN {X 0,Y 198.412,Z 1036.869,A -85,B 0,C 180,E1 -21427.606,E2 -21427.606} C_VEL
LIN {X 0,Y 199.031,Z 1028.151,A -85,B 0,C 180,E1 -21429.913,E2 -21429.913} C_VEL
LIN {X 0,Y 199.687,Z 1018.595,A -85,B 0,C 180,E1 -21431.934,E2 -21431.934} C_VEL
LIN {X 0,Y 200.323,Z 1009.711,A -85,B 0,C 180,E1 -21433.441,E2 -21433.441} C_VEL
LIN {X 0,Y 201.024,Z 999.627,A -85,B 0,C 180,E1 -21434.813,E2 -21434.813} C_VEL
LIN {X 0,Y 201.584,Z 987.455,A -85,B 0,C 180,E1 -21436.066,E2 -21436.066} C_VEL
LIN {X 0,Y 202.563,Z 962.972,A -85,B 0,C 180,E1 -21437.674,E2 -21437.674} C_VEL
LIN {X 0,Y 203.452,Z 933.483,A -85,B 0,C 180,E1 -21439.489,E2 -21439.489} C_VEL
LIN {X 0,Y 200.625,Z 913.612,A -85,B 0,C 180,E1 -21440.734,E2 -21440.734} C_VEL
LIN {X 0,Y 199.939,Z 910.378,A -85,B 0,C 180,E1 -21440.985,E2 -21440.985} C_VEL
LIN {X 0,Y 199.655,Z 910.428,A -85,B 0,C 180,E1 -21444.988,E2 -21444.988} C_VEL
LIN {X 0,Y 199.609,Z 910.429,A -85,B 0,C 180,E1 -21449.534,E2 -21449.534} C_VEL
LIN {X 0,Y 199.667,Z 910.423,A -85,B 0,C 180,E1 -21452.353,E2 -21452.353} C_VEL
LIN {X 0,Y 199.617,Z 910.429,A -85,B 0,C 180,E1 -21456.766,E2 -21456.766} C_VEL
LIN {X 0,Y 199.595,Z 910.43,A -85,B 0,C 180,E1 -21459.333,E2 -21459.333} C_VEL
LIN {X 0,Y 199.567,Z 910.438,A -85,B 0,C 180,E1 -21462.308,E2 -21462.308} C_VEL
LIN {X 0,Y 199.578,Z 910.435,A -85,B 0,C 180,E1 -21465.228,E2 -21465.228} C_VEL
LIN {X 0,Y 199.574,Z 910.434,A -85,B 0,C 180,E1 -21468.004,E2 -21468.004} C_VEL
LIN {X 0,Y 199.599,Z 910.433,A -85,B 0,C 180,E1 -21470.773,E2 -21470.773} C_VEL
LIN {X 0,Y 199.613,Z 910.43,A -85,B 0,C 180,E1 -21475.714,E2 -21475.714} C_VEL
LIN {X 0,Y 199.689,Z 910.418,A -85,B 0,C 180,E1 -21478.135,E2 -21478.135} C_VEL
LIN {X 0,Y 199.647,Z 910.43,A -85,B 0,C 180,E1 -21482.766,E2 -21482.766} C_VEL
LIN {X 0,Y 199.682,Z 910.421,A -85,B 0,C 180,E1 -21487.223,E2 -21487.223} C_VEL
LIN {X 0,Y 199.749,Z 910.414,A -85,B 0,C 180,E1 -21491.803,E2 -21491.803} C_VEL
LIN {X 0,Y 199.814,Z 910.402,A -85,B 0,C 180,E1 -21495.747,E2 -21495.747} C_VEL
LIN {X 0,Y 200.027,Z 910.381,A -85,B 0,C 180,E1 -21499.882,E2 -21499.882} C_VEL
LIN {X 0,Y 200.002,Z 910.381,A -85,B 0,C 180,E1 -21503.949,E2 -21503.949} C_VEL
LIN {X 0,Y 200.266,Z 910.352,A -85,B 0,C 180,E1 -21507.989,E2 -21507.989} C_VEL
LIN {X 0,Y 200.448,Z 910.331,A -85,B 0,C 180,E1 -21510,E2 -21510} C_VEL
LIN {X 0,Y 199.972,Z 910.385,A -85,B 0,C 180,E1 -21514.031,E2 -21514.031} C_VEL
LIN {X 0,Y 200.079,Z 910.374,A -85,B 0,C 180,E1 -21518.077,E2 -21518.077} C_VEL
LIN {X 0,Y 199.86,Z 910.4,A -85,B 0,C 180,E1 -21522.181,E2 -21522.181} C_VEL
LIN {X 0,Y 199.746,Z 910.414,A -85,B 0,C 180,E1 -21526.349,E2 -21526.349} C_VEL
LIN {X 0,Y 199.646,Z 910.428,A -85,B 0,C 180,E1 -21530.612,E2 -21530.612} C_VEL
LIN {X 0,Y 199.625,Z 910.429,A -85,B 0,C 180,E1 -21534.991,E2 -21534.991} C_VEL
LIN {X 0,Y 199.612,Z 910.432,A -85,B 0,C 180,E1 -21539.533,E2 -21539.533} C_VEL
LIN {X 0,Y 199.67,Z 910.419,A -85,B 0,C 180,E1 -21542.352,E2 -21542.352} C_VEL
LIN {X 0,Y 199.622,Z 910.43,A -85,B 0,C 180,E1 -21546.764,E2 -21546.764} C_VEL
LIN {X 0,Y 199.599,Z 910.433,A -85,B 0,C 180,E1 -21549.331,E2 -21549.331} C_VEL
LIN {X 0,Y 199.572,Z 910.435,A -85,B 0,C 180,E1 -21552.307,E2 -21552.307} C_VEL
LIN {X 0,Y 199.58,Z 910.435,A -85,B 0,C 180,E1 -21555.227,E2 -21555.227} C_VEL
LIN {X 0,Y 199.576,Z 910.438,A -85,B 0,C 180,E1 -21558.003,E2 -21558.003} C_VEL
LIN {X 0,Y 199.601,Z 910.429,A -85,B 0,C 180,E1 -21560.772,E2 -21560.772} C_VEL
LIN {X 0,Y 199.614,Z 910.431,A -85,B 0,C 180,E1 -21565.713,E2 -21565.713} C_VEL
LIN {X 0,Y 199.689,Z 910.421,A -85,B 0,C 180,E1 -21568.134,E2 -21568.134} C_VEL
LIN {X 0,Y 199.638,Z 910.43,A -85,B 0,C 180,E1 -21572.763,E2 -21572.763} C_VEL
LIN {X 0,Y 199.671,Z 910.423,A -85,B 0,C 180,E1 -21577.22,E2 -21577.22} C_VEL
LIN {X 0,Y 199.749,Z 910.414,A -85,B 0,C 180,E1 -21581.802,E2 -21581.802} C_VEL
LIN {X 0,Y 199.794,Z 910.408,A -85,B 0,C 180,E1 -21585.744,E2 -21585.744} C_VEL
LIN {X 0,Y 200.026,Z 910.38,A -85,B 0,C 180,E1 -21589.881,E2 -21589.881} C_VEL
LIN {X 0,Y 200,Z 910.384,A -85,B 0,C 180,E1 -21593.948,E2 -21593.948} C_VEL
LIN {X 0,Y 200.264,Z 910.348,A -85,B 0,C 180,E1 -21597.988,E2 -21597.988} C_VEL
LIN {X 0,Y 200.446,Z 910.328,A -85,B 0,C 180,E1 -21599.999,E2 -21599.999} C_VEL
LIN {X 0,Y 199.97,Z 910.389,A -85,B 0,C 180,E1 -21604.03,E2 -21604.03} C_VEL
LIN {X 0,Y 200.072,Z 910.371,A -85,B 0,C 180,E1 -21608.076,E2 -21608.076} C_VEL
LIN {X 0,Y 199.857,Z 910.402,A -85,B 0,C 180,E1 -21612.18,E2 -21612.18} C_VEL
LIN {X 0,Y 199.742,Z 910.412,A -85,B 0,C 180,E1 -21616.348,E2 -21616.348} C_VEL
LIN {X 0,Y 199.642,Z 910.429,A -85,B 0,C 180,E1 -21620.611,E2 -21620.611} C_VEL
LIN {X 0,Y 199.621,Z 910.428,A -85,B 0,C 180,E1 -21624.99,E2 -21624.99} C_VEL
LIN {X 0,Y 199.608,Z 910.434,A -85,B 0,C 180,E1 -21629.532,E2 -21629.532} C_VEL
LIN {X 0,Y 199.666,Z 910.423,A -85,B 0,C 180,E1 -21632.351,E2 -21632.351} C_VEL
LIN {X 0,Y 199.617,Z 910.429,A -85,B 0,C 180,E1 -21636.763,E2 -21636.763} C_VEL
LIN {X 0,Y 199.594,Z 910.434,A -85,B 0,C 180,E1 -21639.33,E2 -21639.33} C_VEL
LIN {X 0,Y 199.567,Z 910.434,A -85,B 0,C 180,E1 -21642.307,E2 -21642.307} C_VEL
LIN {X 0,Y 199.575,Z 910.433,A -85,B 0,C 180,E1 -21645.227,E2 -21645.227} C_VEL
LIN {X 0,Y 199.571,Z 910.439,A -85,B 0,C 180,E1 -21648.002,E2 -21648.002} C_VEL
LIN {X 0,Y 199.596,Z 910.432,A -85,B 0,C 180,E1 -21650.772,E2 -21650.772} C_VEL
